(* CODESYS project plc_chalet_xts.library
   Title: CHALET_Xts
   Version: 4.0.4
   Placeholder: CHALET_Xts
   Company: Beckhoff CH

Project tree, tasks and I/O mapping:
  libraries: CHALET_BaseComponents, * (Beckhoff CH); CHALET_Nc, * (Beckhoff CH); Tc2_EtherCAT, * (Beckhoff Automation GmbH); Tc2_Math, * (Beckhoff Automation GmbH); Tc2_MC2, * (Beckhoff Automation GmbH); Tc2_Standard, * (Beckhoff Automation GmbH); Tc2_System, * (Beckhoff Automation GmbH); Tc3_EventLogger, * (Beckhoff Automation GmbH); Tc3_Mc3Definitions, * (Beckhoff Automation GmbH); Tc3_McCollisionAvoidance, * (Beckhoff Automation GmbH); Tc3_McCoordinatedMotion, * (Beckhoff Automation GmbH); Tc3_Module, * (Beckhoff Automation GmbH); Tc3_XTS_Utility, * (Beckhoff Automation GmbH)
  COMPENENTs/
    Casting/
      function ToEnvironment [ST]
      function ToGroup [ST]
      function ToMover [ST]
      function ToMover_PLC [ST]
      function ToStation [ST]
      function ToStation_PLC [ST]
      function ToTrigger [ST]
    Environment/
      function block FB_XTS_Environment [ST]: FB_init, HR, Initialize, TrackIsRing, TrackLength, Update, UtilityEnvirement
      interface I_XTS_Environment: HR, Initialize, TrackIsRing, TrackLength, Update, UtilityEnvirement
    Group/
      data type E_NcGroupCommands
      function block FB_XTS_Group [ST]: AddAxisListToGroup, AddingAxisToGroup, AllAxesStanding, ChangeGapMode, Disable, Enable, FB_init, GroupEnabled, HR, Initialize, Mapped, OID, RemoveAxisFromGroup, Reset, UngroupAllAxes, Update, UtilityCAGroup
      interface I_XTS_Group: AddAxisListToGroup, AddingAxisToGroup, AllAxesStanding, ChangeGapMode, Disable, Enable, GroupEnabled, HR, Initialize, RemoveAxisFromGroup, Reset, UngroupAllAxes, Update, UtilityCAGroup
    Mover/
      ProductData/
        function block FB_XTS_ProductData [ST]: LinkedMover, LinkToMover
        interface I_XTS_ProductData: LinkedMover, LinkToMover
      function block FB_XTS_Axis [ST]: HaltCA, MoveAbsoluteCA, Update
      function block FB_XTS_Mover [ST]: Disable, Enable, HaltCA, MoveAbsCA, Reset, DefaultAcceleration, DefaultDeceleration, DefaultJerk, SetAcceleration, SetVelocity, Coupled, DrivenDistance, Feedback, getAxisRef, IdentInGroup, LagDistance, LastCmdTargedGap, LastCmdTargedPosition, LastCmdTargedVelocity, MoverInGroup, Moving, NextMover, OID, ParentStation, PositionOnTrack, TargedStation, FB_init, FullAccess, Initialize, ProductData, Update, UtilityMover
      interface I_XTS_Mover: Coupled, Disable, DrivenDistance, Enable, Feedback, getAxisRef, HaltCA, IdentInGroup, LagDistance, LastCmdTargedGap, LastCmdTargedPosition, LastCmdTargedVelocity, MoveAbsCA, MoverInGroup, Moving, NextMover, OID, ParentStation, PositionOnTrack, Reset, SetAcceleration, SetVelocity, TargedStation, UtilityMover
      interface I_XTS_Mover_PLC: DefaultAcceleration, DefaultDeceleration, DefaultJerk, DrivenDistance, FullAccess, LagDistance, LastCmdTargedGap, LUID, PositionOnTrack, ProductData, SetVelocity, TargedStation, UtilityMover
    Station/
      function block FB_XTS_Station [ST]: ChangePos, CtsEmptySpaceInQueue, CtsMoversInQueue, FullAccess, MoverGapAtExit, MoverQueueSize, MoversInPlace, MoversInQueue, MoverVelocityAtExit, PositionOnTrack, SuppressDynamicsChange, TargetPosMonitoringTime, TargetPosWindow, ProcessSimulationActive, Simulation, SimulationMode, MoverPerMin, UpdateStatistic, UpdateUtilityStation, UtilityStationInfo, AddMoverToQueue, DeleteMoversQueue, FB_init, HR, Initialize, OID, Prepare, ReadyToRecvMovers, SendMoversToStation, StationBehinde, StationsAhead, TrySendMoverToNextStation, Update
      interface I_XTS_Station: AddMoverToQueue, CtsEmptySpaceInQueue, CtsMoversInQueue, DeleteMoversQueue, HR, LUID, MoverGapAtExit, MoverQueueSize, MoversInPlace, MoversInQueue, MoverVelocityAtExit, PositionOnTrack, ReadyToRecvMovers, SendMoversToStation, StationsAhead
      interface I_XTS_Station_PLC: ProcessSimulationActive, SimulationMode, ChangePos, FullAccess, LUID, MoverQueueSize, MoversInPlace, MoversInQueue, MoverVelocityAtExit, PositionOnTrack, ReadyToRecvMovers, SendMoversToStation, SuppressDynamicsChange, TargetPosMonitoringTime, TargetPosWindow
    System/
      function block FB_XTS_System [ST]: Disable, Disabled, Disabling, Enable, Enabled, Enabling, Initialize, Initialized, LinkEnvironment, LinkGroup, RegisterMover, RegisterStation, RegisterTrigger, RegisterZone, Environment, Feedback, getMoverInFront, getStationInFront, Movers, Reset, Station, Stations, SuppressAllDynamicsChanges, TrackLength, Triggers, Update, Zones
      interface I_XTS_System_PLC: Disable, Disabled, Enable, Enabled, Feedback, Initialize, Initialized, Reset, Station, SuppressAllDynamicsChanges, TrackLength, Update
      interface I_XTS_System_Registration: Disabled, Enabled, Environment, getMoverInFront, getStationInFront, Initialized, LinkEnvironment, LinkGroup, Movers, RegisterMover, RegisterStation, RegisterTrigger, RegisterZone, Stations, TrackLength
    Trigger/
      function block FB_XTS_Trigger [ST]: FB_init, HR, Initialize, ListOfMoversToCheck, MoverAtTrigger, MoverDetected, PositionOnTrack, Prepare, TimeStamp, TriggerDirection, Update
      interface I_XTS_Trigger: HR, ListOfMoversToCheck, MoverAtTrigger, MoverDetected, PositionOnTrack, TimeStamp, TriggerDirection
    Zone/
      function block FB_XTS_Zone [ST]: CtsMoversInZone, EndPositionOnTrack, FB_init, HR, Initialize, ListOfMoversToCheck, MoversInZone, Prepare, StartPositionOnTrack, Update
      interface I_XTS_Zone: CtsMoversInZone, EndPositionOnTrack, HR, ListOfMoversToCheck, MoversInZone, StartPositionOnTrack
    Class Diagram
  Diag/
    function block FB_XtsEtherCatDiag [ST]: FB_init, Initialize, Initialized, Update
    data type ST_XtsMotorEtherCatDiag
  FUNCTIONs/
    function F_BuildLogString [ST]
    function F_GetDistToPosModulo [ST]
    function F_InLimitTest [ST]
  00000000-0000-0000-0000-000000000000|LICENSE.md
  LICENSE.md
  global variables XtsParameterlist
*)

// COMPENENTs/Group/E_NcGroupCommands
{attribute 'qualified_only'}
{attribute 'strict'}
{attribute 'to_string'}
TYPE E_NcGroupCommands :
(
	None:=0,
	GroupDisable:=150,
	GroupEnable,
	GroupReset,
	AddAxisListToGroup,
	RemoveAxisFromGroup,
	UngroupAllAxes
);
END_TYPE

// Diag/ST_XtsMotorEtherCatDiag
TYPE ST_XtsMotorEtherCatDiag :
STRUCT
	fbSource : FB_TcSourceInfo;
	fbAlarmNotInOpMode : FB_TcAlarm;
	fbAlarmNoCommunication : FB_TcAlarm;
	
	fbGetSlaveState : FB_EcGetSlaveState;
	nLastState : BYTE;
END_STRUCT
END_TYPE

// XtsParameterlist
{attribute 'qualified_only'}
VAR_GLOBAL CONSTANT
	
	(*Checks whether the TC3 event logger is set as standard in the XTS prosessing unit.*)
	B_MSG_IF_TC3EVENTLOGGER_IS_NOT_DEFAULT: BOOL := TRUE;	

	MAX_MOVER_PER_SYSTEM : UINT := 50;
	MAX_MOTORS_PER_SYSTEM : UINT := 100;
	STATISTIC_AVG_PERIOD : TIME := T#10S;
END_VAR

// COMPENENTs/Casting/ToEnvironment
FUNCTION ToEnvironment : BOOL
VAR_INPUT
	ipChObject : I_CH_OBJECT;
	ipXtsEnvironment : REFERENCE TO I_XTS_Environment;
END_VAR

VAR
	ipTmp : I_XTS_Environment;
END_VAR

(* 
   1. Test if the interface exists
   2. Test if the object implements a "Object" interface 
   3. Write reference to interface in parameter
   4. Returne TRUE if succesfull
*)
IF ipChObject <> 0 AND_THEN __QUERYINTERFACE(ipChObject,ipTmp) THEN
	ipXtsEnvironment := ipTmp;
	ToEnvironment := TRUE;
END_IF

END_FUNCTION

// COMPENENTs/Environment/I_XTS_Environment
INTERFACE I_XTS_Environment  EXTENDS I_CH_Object

{attribute 'monitoring':='call'}
PROPERTY HR : HRESULT
GET
END_GET
END_PROPERTY

METHOD Initialize : HRESULT
END_METHOD

{attribute 'monitoring':='call'}
PROPERTY TrackIsRing : BOOL
GET
END_GET
END_PROPERTY

{attribute 'monitoring':='call'}
PROPERTY TrackLength : LREAL
GET
END_GET
END_PROPERTY

METHOD Update : HRESULT
VAR_INPUT
END_VAR
END_METHOD

PROPERTY UtilityEnvirement : Tc3_XTS_Utility.i_TcIoXtsEnvironment
GET
END_GET
END_PROPERTY

END_INTERFACE

// COMPENENTs/Casting/ToGroup
FUNCTION ToGroup : BOOL
VAR_INPUT
	ipChObject : I_CH_OBJECT;
	ipXtsGroup : REFERENCE TO I_XTS_Group;
END_VAR

VAR
	ipTmp : I_XTS_Group;
END_VAR

(* 
   1. Test if the interface exists
   2. Test if the object implements a "Object" interface 
   3. Write reference to interface in parameter
   4. Returne TRUE if succesfull
*)
IF ipChObject <> 0 AND_THEN __QUERYINTERFACE(ipChObject,ipTmp) THEN
	ipXtsGroup := ipTmp;
	ToGroup := TRUE;
END_IF

END_FUNCTION

// COMPENENTs/Group/I_XTS_Group
INTERFACE I_XTS_Group  EXTENDS I_CH_Object

METHOD AddAxisListToGroup : HRESULT
VAR_INPUT
	ipMovers : I_CH_List;
END_VAR
END_METHOD

METHOD AddingAxisToGroup : HRESULT
END_METHOD

PROPERTY AllAxesStanding : Bool
GET
END_GET
END_PROPERTY

METHOD ChangeGapMode : HRESULT
VAR_INPUT
	bFast : BOOL;
END_VAR
END_METHOD

METHOD Disable : HRESULT
VAR_INPUT
END_VAR
END_METHOD

METHOD Enable : HRESULT
VAR_INPUT
END_VAR
END_METHOD

{attribute 'monitoring':='call'}
PROPERTY GroupEnabled : BOOL
GET
END_GET
END_PROPERTY

{attribute 'monitoring':='call'}
PROPERTY HR : HRESULT
GET
END_GET
END_PROPERTY

METHOD Initialize : HRESULT
VAR_INPUT
END_VAR
END_METHOD

METHOD RemoveAxisFromGroup : HRESULT
VAR_INPUT
	ipMover : I_XTS_Mover;
END_VAR
END_METHOD

METHOD Reset : HRESULT
VAR_INPUT
END_VAR
END_METHOD

METHOD UngroupAllAxes : HRESULT
VAR_INPUT
END_VAR
END_METHOD

METHOD Update : HRESULT
VAR_INPUT
END_VAR
END_METHOD

{attribute 'monitoring':='call'}
PROPERTY UtilityCAGroup : I_Mc2CaGroup
GET
END_GET
END_PROPERTY

END_INTERFACE

// COMPENENTs/Mover/I_XTS_Mover
INTERFACE I_XTS_Mover EXTENDS I_CH_Object

{attribute 'OPC.UA.DA.Property' := '1'}
{attribute 'monitoring':='call'}
PROPERTY Coupled : BOOL
GET
END_GET
END_PROPERTY

METHOD Disable : HRESULT
VAR_INPUT
END_VAR
END_METHOD

{attribute 'monitoring':='call'}
PROPERTY DrivenDistance : LREAL
GET
END_GET
END_PROPERTY

METHOD Enable : HRESULT
VAR_INPUT
END_VAR
END_METHOD

{attribute 'OPC.UA.DA.Property' := '1'}
{attribute 'monitoring':='call'}
PROPERTY Feedback : I_CH_Feedback
GET
END_GET
END_PROPERTY

PROPERTY getAxisRef : REFERENCE TO Tc2_MC2.AXIS_REF
GET
END_GET
END_PROPERTY

METHOD HaltCA : HRESULT
VAR_INPUT
END_VAR
END_METHOD

{attribute 'monitoring':='call'}
PROPERTY IdentInGroup : IDENT_IN_GROUP_REF
GET
END_GET
END_PROPERTY

{attribute 'monitoring':='call'}
PROPERTY LagDistance : LREAL
GET
END_GET
END_PROPERTY

{attribute 'monitoring':='call'}
PROPERTY LastCmdTargedGap : LREAL
GET
END_GET
END_PROPERTY

{attribute 'monitoring':='call'}
PROPERTY LastCmdTargedPosition : LREAL
GET
END_GET
END_PROPERTY

{attribute 'monitoring':='call'}
PROPERTY LastCmdTargedVelocity : LREAL
GET
END_GET
END_PROPERTY

METHOD MoveAbsCA : HRESULT
VAR_INPUT
    fPosition              : LREAL;
    fVelocity              : LREAL;
    fGap                   : LREAL;
    eDirection             : Tc3_Mc3Definitions.MC_DIRECTION;
END_VAR
END_METHOD

{attribute 'monitoring':='call'}
PROPERTY MoverInGroup : BOOL
GET
END_GET
SET
END_SET
END_PROPERTY

{attribute 'OPC.UA.DA.Property' := '1'}
{attribute 'monitoring':='call'}
PROPERTY Moving : BOOL
GET
END_GET
END_PROPERTY

{attribute 'monitoring':='call'}
PROPERTY NextMover : I_XTS_Mover
GET
END_GET
END_PROPERTY

{attribute 'monitoring':='call'}
PROPERTY OID : OTCID
GET
END_GET
END_PROPERTY

{attribute 'monitoring':='call'}
PROPERTY ParentStation : I_XTS_Station
GET
END_GET
SET
END_SET
END_PROPERTY

{attribute 'monitoring':='call'}
PROPERTY PositionOnTrack : LREAL
GET
END_GET
END_PROPERTY

METHOD Reset : HRESULT
VAR_INPUT
END_VAR
END_METHOD

{attribute 'monitoring':='call'}
PROPERTY SetAcceleration : LREAL
GET
END_GET
END_PROPERTY

{attribute 'monitoring':='call'}
PROPERTY SetVelocity : LREAL
GET
END_GET
END_PROPERTY

{attribute 'monitoring':='call'}
PROPERTY TargedStation : STRING
GET
END_GET
SET
END_SET
END_PROPERTY

{attribute 'monitoring':='call'}
PROPERTY UtilityMover : I_TcIoXtsXpuMover
GET
END_GET
END_PROPERTY

END_INTERFACE

// COMPENENTs/Station/I_XTS_Station
INTERFACE I_XTS_Station EXTENDS I_CH_Object

METHOD AddMoverToQueue : HRESULT
VAR_INPUT
	ipMover : I_XTS_Mover;
END_VAR
END_METHOD

{attribute 'monitoring':='call'}
PROPERTY CtsEmptySpaceInQueue : UDINT
GET
END_GET
END_PROPERTY

{attribute 'monitoring':='call'}
PROPERTY CtsMoversInQueue : UDINT
GET
END_GET
END_PROPERTY

METHOD DeleteMoversQueue : HRESULT
VAR_INPUT
END_VAR
END_METHOD

{attribute 'monitoring':='call'}
PROPERTY HR : HRESULT
GET
END_GET
END_PROPERTY

{attribute 'monitoring':='call'}
PROPERTY LUID : STRING
GET
END_GET
END_PROPERTY

{attribute 'monitoring':='call'}
PROPERTY MoverGapAtExit : LREAL
GET
END_GET
END_PROPERTY

{attribute 'monitoring':='call'}
PROPERTY MoverQueueSize : UINT
GET
END_GET
SET
END_SET
END_PROPERTY

{attribute 'monitoring':='call'}
PROPERTY MoversInPlace : BOOL
GET
END_GET
END_PROPERTY

{attribute 'monitoring':='call'}
PROPERTY MoversInQueue : REFERENCE TO ARRAY [0..(XtsParameterlist.MAX_MOVER_PER_SYSTEM-1)] OF I_XTS_Mover_PLC // Return a sorted list of movers in this zone. Index 0 is the mover in Front.
GET
END_GET
END_PROPERTY

{attribute 'monitoring':='call'}
PROPERTY MoverVelocityAtExit : LREAL
GET
END_GET
SET
END_SET
END_PROPERTY

{attribute 'monitoring':='call'}
PROPERTY PositionOnTrack : LREAL
GET
END_GET
END_PROPERTY

{attribute 'monitoring':='call'}
PROPERTY ReadyToRecvMovers : BOOL
GET
END_GET
SET
END_SET
END_PROPERTY

METHOD SendMoversToStation : HRESULT
VAR_INPUT
	sTargedStation : STRING;
END_VAR
END_METHOD

{attribute 'monitoring':='call'}
PROPERTY StationsAhead : I_XTS_Station
GET
END_GET
END_PROPERTY

END_INTERFACE

// COMPENENTs/Mover/I_XTS_Mover_PLC
INTERFACE I_XTS_Mover_PLC EXTENDS I_CH_Object

{attribute 'OPC.UA.DA.Property' := '1'}
{attribute 'monitoring':='call'}
PROPERTY DefaultAcceleration : LREAL
GET
END_GET
SET
END_SET
END_PROPERTY

{attribute 'OPC.UA.DA.Property' := '1'}
{attribute 'monitoring':='call'}
PROPERTY DefaultDeceleration : LREAL
GET
END_GET
SET
END_SET
END_PROPERTY

{attribute 'OPC.UA.DA.Property' := '1'}
{attribute 'monitoring':='call'}
PROPERTY DefaultJerk : LREAL
GET
END_GET
SET
END_SET
END_PROPERTY

{attribute 'monitoring':='call'}
PROPERTY DrivenDistance : LREAL
GET
END_GET
END_PROPERTY

(*The _ PLC interface provides the user with a simplified interface for commanding between the stations. Sometimes, however, this is not enough. 
Either you get the corresponding interface with the __Queryinterface or you can get full access with this property.*)
PROPERTY FullAccess : I_XTS_Mover
GET
END_GET
END_PROPERTY

{attribute 'monitoring':='call'}
PROPERTY LagDistance : LREAL
GET
END_GET
END_PROPERTY

{attribute 'monitoring':='call'}
PROPERTY LastCmdTargedGap : LREAL
GET
END_GET
END_PROPERTY

{attribute 'monitoring':='call'}
PROPERTY LUID : STRING
GET
END_GET
END_PROPERTY

{attribute 'monitoring':='call'}
PROPERTY PositionOnTrack : LREAL
GET
END_GET
END_PROPERTY

{attribute 'monitoring':='call'}
PROPERTY PUBLIC ProductData : I_XTS_ProductData
GET
END_GET
SET
END_SET
END_PROPERTY

{attribute 'monitoring':='call'}
PROPERTY SetVelocity : LREAL
GET
END_GET
END_PROPERTY

{attribute 'monitoring':='call'}
PROPERTY TargedStation : STRING
GET
END_GET
END_PROPERTY

{attribute 'monitoring':='call'}
PROPERTY UtilityMover : I_TcIoXtsXpuMover
GET
END_GET
END_PROPERTY

END_INTERFACE

// COMPENENTs/Mover/ProductData/I_XTS_ProductData
INTERFACE I_XTS_ProductData EXTENDS __SYSTEM.IQueryInterface

{attribute 'monitoring':='call'}
PROPERTY LinkedMover : I_XTS_Mover_PLC
GET
END_GET
END_PROPERTY

METHOD LinkToMover : BOOL //it is not necessary to call this method. This is already done internally
VAR_INPUT
	ipMoverPlc : I_XTS_Mover_PLC;
END_VAR
END_METHOD

END_INTERFACE

// COMPENENTs/Casting/ToMover
FUNCTION ToMover : BOOL
VAR_INPUT
	ipChObject : I_CH_OBJECT;
	ipXtsMover : REFERENCE TO I_XTS_Mover;
END_VAR

VAR
	ipTmp : I_XTS_Mover;
END_VAR

(* 
   1. Test if the interface exists
   2. Test if the object implements a "Object" interface 
   3. Write reference to interface in parameter
   4. Returne TRUE if succesfull
*)
IF ipChObject <> 0 AND_THEN __QUERYINTERFACE(ipChObject,ipTmp) THEN
	ipXtsMover := ipTmp;
	ToMover := TRUE;
END_IF

END_FUNCTION

// COMPENENTs/Casting/ToMover_PLC
FUNCTION ToMover_PLC : BOOL
VAR_INPUT
	ipChObject : I_CH_OBJECT;
	ipXtsMover : REFERENCE TO I_XTS_Mover_PLC;
END_VAR

VAR
	ipTmp : I_XTS_Mover_PLC;
END_VAR

(* 
   1. Test if the interface exists
   2. Test if the object implements a "Object" interface 
   3. Write reference to interface in parameter
   4. Returne TRUE if succesfull
*)
IF ipChObject <> 0 AND_THEN __QUERYINTERFACE(ipChObject,ipTmp) THEN
	ipXtsMover := ipTmp;
	ToMover_PLC := TRUE;
END_IF

END_FUNCTION

// COMPENENTs/Casting/ToStation
FUNCTION ToStation : BOOL
VAR_INPUT
	ipChObject : I_CH_OBJECT;
	ipXtsStation : REFERENCE TO I_XTS_Station;
END_VAR

VAR
	ipTmp : I_XTS_Station;
END_VAR

(* Register the Station
   1. Test if the interface exists
   2. Test if the object implements a "Object" interface 
*)
IF ipChObject <> 0 AND_THEN __QUERYINTERFACE(ipChObject,ipTmp) THEN
	ipXtsStation := ipTmp;
	ToStation := TRUE;
END_IF

END_FUNCTION

// COMPENENTs/Casting/ToStation_PLC
FUNCTION ToStation_PLC : BOOL
VAR_INPUT
	ipChObject : I_CH_OBJECT;
	ipXtsStationPLC : REFERENCE TO I_XTS_Station_PLC;
END_VAR

VAR
	ipTmp : I_XTS_Station_PLC;
END_VAR

(* Register the Station
   1. Test if the interface exists
   2. Test if the object implements a "Object" interface 
*)
IF ipChObject <> 0 AND_THEN __QUERYINTERFACE(ipChObject,ipTmp) THEN
	ipXtsStationPLC := ipTmp;
	ToStation_PLC := TRUE;
END_IF

END_FUNCTION

// COMPENENTs/Station/I_XTS_Station_PLC
INTERFACE I_XTS_Station_PLC EXTENDS I_CH_Object

{attribute 'monitoring':='call'}
PROPERTY ProcessSimulationActive : BOOL
GET
END_GET
END_PROPERTY

//If a valid time (>0seconds) is set and the configured destination station exists, then the movers will be sent away automatically after this time from now on.
METHOD SimulationMode : HRESULT
VAR_INPUT
	fProcessDuration 	: LREAL; //[s]
	sTargedStation		: STRING; //LUID of the targed station to automatic send after the duration
END_VAR
END_METHOD

METHOD ChangePos : HRESULT
VAR_INPUT
	fNewPosOnTrack : LREAL;
END_VAR
END_METHOD

(*The _ PLC interface provides the user with a simplified interface for commanding between the stations. Sometimes, however, this is not enough. 
Either you get the corresponding interface with the __Queryinterface or you can get full access with this property.*)
PROPERTY FullAccess : I_XTS_Station
GET
END_GET
END_PROPERTY

{attribute 'monitoring':='call'}
PROPERTY LUID : STRING
GET
END_GET
END_PROPERTY

{attribute 'monitoring':='call'}
PROPERTY MoverQueueSize : UINT
GET
END_GET
SET
END_SET
END_PROPERTY

{attribute 'monitoring':='call'}
PROPERTY MoversInPlace : BOOL
GET
END_GET
END_PROPERTY

{attribute 'monitoring':='call'}
PROPERTY MoversInQueue : REFERENCE TO ARRAY [0..(XtsParameterlist.MAX_MOVER_PER_SYSTEM-1)] OF I_XTS_Mover_PLC // Return a sorted list of movers in this zone. Index 0 is the mover in Front.
GET
END_GET
END_PROPERTY

{attribute 'monitoring':='call'}
PROPERTY MoverVelocityAtExit : LREAL //[mm/s] Every mover that leaves or passes the station gets this new velocity as a target.
GET
END_GET
SET
END_SET
END_PROPERTY

{attribute 'monitoring':='call'}
PROPERTY PositionOnTrack : LREAL
GET
END_GET
END_PROPERTY

{attribute 'monitoring':='call'}
//prevent further movers from entering the station, 
//e.g. to prevent a collision. All movers that are already moving to reach this station will be stopped with a stop 
//and restarted with Ready True.
PROPERTY ReadyToRecvMovers : BOOL
GET
END_GET
SET
END_SET
END_PROPERTY

METHOD SendMoversToStation : HRESULT
VAR_INPUT
	sTargedStation : STRING;
END_VAR
END_METHOD

{attribute 'monitoring':='call'}
PROPERTY SuppressDynamicsChange : BOOL
GET
END_GET
SET
END_SET
END_PROPERTY

{attribute 'monitoring':='call'}
//A time that is waited as soon as the mover is in the station (including the monitoring window) before “MoversInPlace” is set. e.g. used to stabilize the workpiece
PROPERTY TargetPosMonitoringTime : TIME
GET
END_GET
SET
END_SET
END_PROPERTY

{attribute 'monitoring':='call'}
//How many mm before the mover reaches the position is “MoversInPlace” set for the process. 
//This distance can also be set very large (e.g. 100mm) for moving past without stopping.
PROPERTY TargetPosWindow : LREAL
GET
END_GET
SET
END_SET
END_PROPERTY

END_INTERFACE

// COMPENENTs/Casting/ToTrigger
FUNCTION ToTrigger : BOOL
VAR_INPUT
	ipChObject : I_CH_OBJECT;
	ipXtsTrigger : REFERENCE TO I_XTS_Trigger;
END_VAR

VAR
	ipTmp : I_XTS_Trigger;
END_VAR

(* 
   1. Test if the interface exists
   2. Test if the object implements a "Object" interface 
   3. Write reference to interface in parameter
   4. Returne TRUE if succesfull
*)
IF ipChObject <> 0 AND_THEN __QUERYINTERFACE(ipChObject,ipTmp) THEN
	ipXtsTrigger := ipTmp;
	ToTrigger := TRUE;
END_IF

END_FUNCTION

// COMPENENTs/Trigger/I_XTS_Trigger
INTERFACE I_XTS_Trigger  EXTENDS I_CH_Object

{attribute 'monitoring':='call'}
PROPERTY HR : HRESULT
GET
END_GET
END_PROPERTY

PROPERTY ListOfMoversToCheck : I_CH_List
SET
END_SET
END_PROPERTY

{attribute 'monitoring':='call'}
PROPERTY MoverAtTrigger : I_XTS_Mover
GET
END_GET
END_PROPERTY

{attribute 'monitoring':='call'}
PROPERTY MoverDetected : BOOL
GET
END_GET
END_PROPERTY

{attribute 'monitoring':='call'}
PROPERTY PositionOnTrack : LREAL
GET
END_GET
SET
END_SET
END_PROPERTY

{attribute 'monitoring':='call'}
PROPERTY TimeStamp : T_DCTIME64;
GET
END_GET
END_PROPERTY

{attribute 'monitoring':='call'}
PROPERTY TriggerDirection : Tc2_MC2.MC_Direction
GET
END_GET
SET
END_SET
END_PROPERTY

END_INTERFACE

// COMPENENTs/Environment/FB_XTS_Environment
{attribute 'no_explicit_call' := 'Do not call the body - Stick to OOP'}
FUNCTION_BLOCK FB_XTS_Environment EXTENDS FB_CH_Object IMPLEMENTS I_XTS_Environment
VAR
	{attribute 'hide'}
	bInitDone : BOOL ;
	{attribute 'hide'}
	ipXtsSystem : I_XTS_System_Registration;

	fbUtilityEnvironment : Tc3_XTS_Utility.FB_TcIoXtsEnvironment;
	
	//Ethercat Diagnostic of all XTS Motors
	fbXtsEtherCatDiag		: FB_XtsEtherCatDiag(	ipUtilityEnvironmentv 				:=  fbUtilityEnvironment,
													bCheckIfTc3EventloggerIsSelected 	:= XtsParameterlist.B_MSG_IF_TC3EVENTLOGGER_IS_NOT_DEFAULT);
	
	{attribute 'hide'}
	fbXtsEnvironmentVisu : Tc3_XTS_Utility.FB_XtsEnvironmentVisu;
		
END_VAR

METHOD FB_init : BOOL
VAR_INPUT
	bInitRetains : BOOL; // if TRUE, the retain variables are initialized (warm start / cold start)
	bInCopyCode : BOOL;  // if TRUE, the instance afterwards gets moved into the copy code (online change)

	ipXtsSystem : I_XTS_System_Registration; //Interface to XTS system object	
END_VAR
VAR_INST
	{attribute 'hide'}
	bFBInitCalledOnce : BOOL; //Do the following code once during start up and not during onlinechange
END_VAR
//Do the following code once during start up and not during onlinechange
IF NOT bFBInitCalledOnce THEN 
	
	//Regristrate object in System
	IF ipXtsSystem <> 0 THEN
		ipXtsSystem.LinkEnvironment(THIS^);
		THIS^.ipXtsSystem := ipXtsSystem;
	END_IF



END_IF

bFBInitCalledOnce := TRUE;
END_METHOD

{warning 'add property implementation'}
{attribute 'monitoring':='call'}
PROPERTY HR : HRESULT
GET
HR := S_OK;
END_GET
END_PROPERTY

METHOD Initialize : HRESULT
VAR 
	hr : HRESULT;
END_VAR
IF NOT THIS^.bInitDone THEN
	Initialize := S_PENDING;	

	//Enable init Info Server if needed
	fbUtilityEnvironment.P_XtsEnvironmentConfiguration.bEnableInitInfoServer := TRUE;

	//Enable init CA Group if needed
	fbUtilityEnvironment.P_XtsEnvironmentConfiguration.bEnableInitCaGroup := TRUE;

	IF NOT fbUtilityEnvironment.P_IsInitialized THEN	
		//Start init
		fbUtilityEnvironment.Init(bExecute := TRUE); 
		hr := GetMostSignificant(hr, S_PENDING);	
 	ELSE
		//Stop init
		fbUtilityEnvironment.Init(bExecute := FALSE);
	END_IF
	
	// Link data Pointer 
	fbXtsEnvironmentVisu(ipTcIoXtsEnvironment:=UtilityEnvirement);

	// Ethercat Diagnostic of all XTS Motors
	hr := GetMostSignificant(hr, fbXtsEtherCatDiag.Initialize());
	

	THIS^.bInitDone  :=  hr = S_OK;
END_IF

Initialize := hr;
END_METHOD

{attribute 'monitoring':='call'}
PROPERTY TrackIsRing : BOOL
GET
IF fbUtilityEnvironment.P_IsInitialized THEN
	TrackIsRing := fbUtilityEnvironment.Mc2CaGroup(1).GetRailIsRing();
END_IF
END_GET
END_PROPERTY

{attribute 'monitoring':='call'}
PROPERTY TrackLength : LREAL
GET
IF fbUtilityEnvironment.P_IsInitialized THEN
	TrackLength := fbUtilityEnvironment.Mc2CaGroup(1).GetRailLength();
END_IF
END_GET
END_PROPERTY

METHOD Update : HRESULT
VAR
	hr : HRESULT;
END_VAR

fbXtsEtherCatDiag.Update();

fbXtsEnvironmentVisu.Cycle();

Update:= hr;
END_METHOD

PROPERTY UtilityEnvirement : Tc3_XTS_Utility.I_TcIoXtsEnvironment
GET
//Interface to envirement
UtilityEnvirement := fbUtilityEnvironment;
END_GET
END_PROPERTY

END_FUNCTION_BLOCK

// COMPENENTs/System/I_XTS_System_Registration
INTERFACE I_XTS_System_Registration

{attribute 'monitoring':='call'}
PROPERTY Disabled : Bool
GET
END_GET
END_PROPERTY

{attribute 'monitoring':='call'}
PROPERTY Enabled : Bool
GET
END_GET
END_PROPERTY

{attribute 'monitoring':='call'}
PROPERTY Environment : I_XTS_Environment
GET
END_GET
END_PROPERTY

METHOD getMoverInFront : I_Xts_Mover
VAR_INPUT
	ipMover : I_Xts_Mover;
END_VAR
END_METHOD

METHOD getStationInFront : I_XTS_Station
VAR_INPUT
	ipStation : I_XTS_Station;
END_VAR
END_METHOD

{attribute 'monitoring':='call'}
PROPERTY Initialized : BOOL
GET
END_GET
END_PROPERTY

METHOD LinkEnvironment : HRESULT
VAR_INPUT
	ipEnvironment : CHALET_BaseComponents.I_CH_Object;
END_VAR
END_METHOD

METHOD LinkGroup : HRESULT
VAR_INPUT
	ipGroup : CHALET_BaseComponents.I_CH_Object;
END_VAR
END_METHOD

{attribute 'monitoring':='call'}
PROPERTY Movers : CHALET_BaseComponents.I_CH_LIST
GET
END_GET
END_PROPERTY

METHOD RegisterMover : HRESULT
VAR_INPUT
	ipMover : CHALET_BaseComponents.I_CH_Object;
END_VAR
END_METHOD

METHOD RegisterStation : HRESULT
VAR_INPUT
	ipStation : CHALET_BaseComponents.I_CH_Object;
END_VAR
END_METHOD

METHOD RegisterTrigger : HRESULT
VAR_INPUT
	ipTrigger	: CHALET_BaseComponents.I_CH_Object;
END_VAR
END_METHOD

METHOD RegisterZone : HRESULT
VAR_INPUT
	ipZone	: CHALET_BaseComponents.I_CH_Object;
END_VAR
END_METHOD

PROPERTY Stations : I_CH_LIST
GET
END_GET
END_PROPERTY

{attribute 'monitoring':='call'}
PROPERTY TrackLength : LREAL
GET
END_GET
END_PROPERTY

END_INTERFACE

// Diag/FB_XtsEtherCatDiag
{attribute 'no_explicit_call' := 'Do not call the body - Stick to OOP'}
(* This FB generates an array with all XTS motor modules. These are now checked cyclically one after the other to see whether the EtherCAT slave controller is in OP mode *)
FUNCTION_BLOCK FB_XtsEtherCatDiag EXTENDS CHALET_BaseComponents.FB_CH_Object
VAR
	ipUtilityEnvironmentv : Tc3_XTS_Utility.I_TcIoXtsEnvironment;
	bCheckIfTc3EventloggerIsSelected : BOOL;
	stMotorDiag : ARRAY[0..N_MAX_CTS_MOTORMODULES-1] OF ST_XtsMotorEtherCatDiag;
	bInitDone : BOOL;
	nIdxTrigger : UINT;
	nCtnMotorModules : UINT;
	fbMsgWrongEventlogger : FB_TcMessage;
	bEventLoggerChecked : BOOL;
END_VAR

VAR CONSTANT
	N_MAX_CTS_MOTORMODULES : UINT := XtsParameterlist.MAX_MOTORS_PER_SYSTEM;
END_VAR

METHOD FB_init : BOOL
VAR_INPUT
	bInitRetains : BOOL; // if TRUE, the retain variables are initialized (warm start / cold start)
	bInCopyCode : BOOL;  // if TRUE, the instance afterwards gets moved into the copy code (online change)
	
	ipUtilityEnvironmentv : Tc3_XTS_Utility.I_TcIoXtsEnvironment;
	
	//Message if TC3_Eventlogger is not set as Eventlogger. Not possible to change online.
	//Must be adjusted in the following object: XtsProcessingUnit/Parameter(Init)/Diagnostic/UsedEventLogger 
	bCheckIfTc3EventloggerIsSelected : BOOL;
END_VAR

VAR
	fbGetCurTaskIdx  : GETCURTASKINDEX;
END_VAR

THIS^.ipUtilityEnvironmentv := ipUtilityEnvironmentv;
THIS^.bCheckIfTc3EventloggerIsSelected := bCheckIfTc3EventloggerIsSelected;
END_METHOD

METHOD Initialize : HRESULT
VAR
	ipObject : ITComObject;
	sObjectName : STRING;
	nIdx, nIdxXpu, nIdxPart, nIdxModule : UINT;
END_VAR
VAR_INST

END_VAR
//Validate interface
IF ipUtilityEnvironmentv = 0 THEN
	Initialize := E_FAIL;
	RETURN;
END_IF

//Wait for an valide XpuCount. At beginn, count is 0
IF ipUtilityEnvironmentv.P_XpuCount = 0 THEN
	Initialize := S_PENDING;;
	RETURN;
END_IF

//Wait for init done
FOR nIdxXpu := 1 TO TO_UINT(ipUtilityEnvironmentv.P_XpuCount)  DO
	IF NOT ipUtilityEnvironmentv.XpuTcIo(nIdxXpu).P_IsInitialized THEN
		Initialize := S_PENDING;;
		RETURN;
	END_IF
END_FOR

//Message if TC3_Eventlogger is not set as Eventlogger. Not possible to change online.
//Must be adjusted in the following object: XtsProcessingUnit/Parameter(Init)/Diagnostic/UsedEventLogger 
IF NOT bEventLoggerChecked  AND THIS^.bCheckIfTc3EventloggerIsSelected THEN
	FOR nIdxXpu := 1 TO TO_UINT(ipUtilityEnvironmentv.P_XpuCount) DO
		IF ipUtilityEnvironmentv.XpuTcIo(nIdxXpu).GetUsedEventLogger() <> EventMessenger.TC3EventLogger THEN
			fbMsgWrongEventlogger.CreateEx(stEventEntry:=TC_EVENTS.CHALET_XTS_Events.TC3EventloggerCheck, ipSourceInfo := THIS^.fbSourceInfo);
			fbMsgWrongEventlogger.Send(0);
			EXIT;
		END_IF
	END_FOR
END_IF
bEventLoggerChecked := TRUE;



//For all Modul in all Parts in all Processing-Units
nIdx := 0;
FOR nIdxXpu := 1 TO TO_UINT(ipUtilityEnvironmentv.P_XpuCount) DO
	FOR nIdxPart := 1 TO ipUtilityEnvironmentv.XpuTcIo(nIdxXpu).P_PartCount DO
		FOR nIdxModule := 1 TO ipUtilityEnvironmentv.XpuTcIo(nIdxXpu).PartTcIo(nIdxPart).P_ModuleCount DO
			//Error, array is to small
			IF (nIdx > (N_MAX_CTS_MOTORMODULES-1)) THEN
				Initialize := E_FAIL;
				RETURN;
			END_IF
			
			//Read object name of motor module
			FW_ObjMgr_GetObjectInstance(oid:= ipUtilityEnvironmentv.XpuTcIo(nIdxXpu).PartTcIo(nIdxPart).ModuleTcIo(nIdxModule).GetMotorTerminalOid() , iid:= TC_GLOBAL_IID_LIST.IID_ITComObject, pipUnk:= ADR(ipObject));
			//Read Name of object if interafce is valid
			IF ipObject <> 0 AND_THEN (ipObject.TcGetObjectName(ADR(sObjectName), SIZEOF(sObjectName)) = S_OK) THEN
				//Set source name + Modulename
				stMotorDiag[nIdx].fbSource.sName := '';
				stMotorDiag[nIdx].fbSource.ExtendName(sObjectName);
				stMotorDiag[nIdx].fbSource.ExtendName(' Part:');
				stMotorDiag[nIdx].fbSource.ExtendName(TO_STRING(nIdxPart));
				stMotorDiag[nIdx].fbSource.ExtendName(' Module:');
				stMotorDiag[nIdx].fbSource.ExtendName(TO_STRING(nIdxModule));	
				ipObject.TcRelease();
			ELSE
				//Set source name
				stMotorDiag[nIdx].fbSource.sName := '';
				stMotorDiag[nIdx].fbSource.ExtendName('Part:');
				stMotorDiag[nIdx].fbSource.ExtendName(TO_STRING(nIdxPart));
				stMotorDiag[nIdx].fbSource.ExtendName(' Module:');
				stMotorDiag[nIdx].fbSource.ExtendName(TO_STRING(nIdxModule));	
			END_IF
			

		
			//Create alarm
			stMotorDiag[nIdx].fbAlarmNotInOpMode.CreateEx(
					stEventEntry := TC_EVENTS.CHALET_XTS_Events.EtherCatSlaveNotInOpMode, 
					ipSourceInfo := stMotorDiag[nIdx].fbSource, 
					bWithConfirmation := FALSE);
					
			stMotorDiag[nIdx].fbAlarmNoCommunication.CreateEx(	
					stEventEntry:= TC_EVENTS.CHALET_XTS_Events.NoCommunication,
					ipSourceInfo 	:= stMotorDiag[nIdx].fbSource, 
					bWithConfirmation := FALSE);
					
			//store ADS conncetion info
			stMotorDiag[nIdx].fbGetSlaveState.sNetId := ipUtilityEnvironmentv.XpuTcIo(nIdxXpu).PartTcIo(nIdxPart).ModuleTcIo(nIdxModule).CoE.AmsNetId;
			stMotorDiag[nIdx].fbGetSlaveState.nSlaveAddr := ipUtilityEnvironmentv.XpuTcIo(nIdxXpu).PartTcIo(nIdxPart).ModuleTcIo(nIdxModule).GetDriveAddress();		

			nIdx := nIdx +1;	
			THIS^.nCtnMotorModules := nIdx;
		END_FOR
	END_FOR
END_FOR
bInitDone := TRUE;
Initialize := S_OK;;
END_METHOD

{attribute 'monitoring':='call'}
PROPERTY Initialized : BOOL
GET
Initialized := bInitDone;
END_GET
END_PROPERTY

METHOD Update : HRESULT
VAR
	nIdx : UINT;
	bErrorNoCom : BOOL;
	bInOpMode : BOOL;
	bReadOfStateFailed : BOOL;
END_VAR
// Force to do init
IF NOT THIS^.bInitDone THEN
	Initialize();
	RETURN;
END_IF


//Trigger each plc cycle 1 read of the motor ethercat slave state - if not allready busy
IF NOT stMotorDiag[nIdxTrigger].fbGetSlaveState.bBusy THEN
	stMotorDiag[nIdxTrigger].fbGetSlaveState(bExecute := TRUE);
	stMotorDiag[nIdxTrigger].fbGetSlaveState(bExecute := FALSE);
	nIdxTrigger := (nIdxTrigger + 1)MOD THIS^.nCtnMotorModules;
END_IF



//For all FBs
FOR nIdx := 0 TO (THIS^.nCtnMotorModules-1) DO
	(*	0x___1 = Slave in 'INIT' state
		0x___2 = Slave in 'PREOP' state
		0x___3 = Slave in 'BOOT' state
		0x___4 = Slave in 'SAFEOP' state
		0x___8 = Slave in 'OP' state		*)
		
		
	//Write Ethercat linkState in TC3 Eventlogger
	bErrorNoCom := (stMotorDiag[nIdx].fbGetSlaveState.state.linkState = 16#01(*NotPresent*));
	IF (NOT bErrorNoCom AND stMotorDiag[nIdx].fbAlarmNoCommunication.bRaised) THEN
		//No error - Reset	
		stMotorDiag[nIdx].fbAlarmNoCommunication.Clear(0,0);
	ELSIF (bErrorNoCom AND NOT stMotorDiag[nIdx].fbAlarmNoCommunication.bRaised) THEN
		//New Error - Raise
		stMotorDiag[nIdx].fbAlarmNoCommunication.ipArguments.Clear();
		stMotorDiag[nIdx].fbAlarmNoCommunication.Raise(0);
	ELSE
		//Alarm is already active
		;
	END_IF	

		
	//Re-Raise alarm on change of state if ethercatslave is not in OP-Mode - Clear if NoCommunication is raised
	bInOpMode := (stMotorDiag[nIdx].fbGetSlaveState.state.deviceState = 16#08(*OP*));
	bReadOfStateFailed := ((stMotorDiag[nIdx].fbGetSlaveState.state.deviceState AND 16#0F(*Mask values 0-15*)) = 16#00);
	IF ((bInOpMode OR bErrorNoCom OR bReadOfStateFailed) AND stMotorDiag[nIdx].fbAlarmNotInOpMode.bRaised) THEN
		//No error - Reset	
		stMotorDiag[nIdx].fbAlarmNotInOpMode.Clear(0,0);
		
	ELSIF (bInOpMode OR bErrorNoCom OR bReadOfStateFailed) THEN
		; //Do nothing
		
	ELSIF (stMotorDiag[nIdx].fbGetSlaveState.state.deviceState <> stMotorDiag[nIdx].nLastState) THEN
		//New Error - Reset, Create and Raise
		stMotorDiag[nIdx].fbAlarmNotInOpMode.Clear(0,0);
		CASE (stMotorDiag[nIdx].fbGetSlaveState.state.deviceState AND 16#0F(*Mask values 0-15*)) OF
			1:  stMotorDiag[nIdx].fbAlarmNotInOpMode.ipArguments.Clear().AddString('INIT'); 	
			2:  stMotorDiag[nIdx].fbAlarmNotInOpMode.ipArguments.Clear().AddString('PREOP');	
			3:  stMotorDiag[nIdx].fbAlarmNotInOpMode.ipArguments.Clear().AddString('BOOT');		
			4:  stMotorDiag[nIdx].fbAlarmNotInOpMode.ipArguments.Clear().AddString('SAFEOP');	
		END_CASE
		stMotorDiag[nIdx].fbAlarmNotInOpMode.Raise(0);
		
	ELSE
		//Alarm is already active
		;
	END_IF
	stMotorDiag[nIdx].nLastState := stMotorDiag[nIdx].fbGetSlaveState.state.deviceState;

	
	//Call cyclic fb
	stMotorDiag[nIdx].fbGetSlaveState();
END_FOR
END_METHOD

END_FUNCTION_BLOCK

// COMPENENTs/Group/FB_XTS_Group
{attribute 'no_explicit_call' := 'Do not call the body - Stick to OOP'}
FUNCTION_BLOCK FB_XTS_Group EXTENDS FB_CH_Object IMPLEMENTS I_XTS_Group
VAR
	{attribute 'hide'}	
	bInitDone : BOOL;
	{attribute 'hide'}
	ipXtsSystem 		: I_XTS_System_Registration;
	{attribute 'hide'}
	ipUtilityCAGroup 	: I_Mc2CaGroup;
	{attribute 'hide'}
	fbAddAxisToGroup 	: Tc3_McCoordinatedMotion.MC_AddAxisToGroup;
	{attribute 'hide'}
	fbRemoveAxisToGroup : Tc3_McCoordinatedMotion.MC_RemoveAxisFromGroup;
	{attribute 'hide'}
	fbGroupEnable 		: Tc3_McCoordinatedMotion.MC_GroupEnable;
	{attribute 'hide'}
	fbGroupDisable 		: Tc3_McCoordinatedMotion.MC_GroupDisable;
	{attribute 'hide'}
	fbGroupReadStatus 	: Tc3_McCoordinatedMotion.MC_GroupReadStatus;	
	{attribute 'hide'}
	fbUngroupAllAxes 	: Tc3_McCoordinatedMotion.MC_UngroupAllAxes;	
	{attribute 'hide'}
	fbGroupReset	 	: Tc3_McCoordinatedMotion.MC_GroupReset;
	{attribute 'hide'}
	nState_SEQ_Adding 	: UDINT;
	{attribute 'hide'}	
	fbMovers : CHALET_BaseComponents.FB_CH_List; // List of Axis to be added to the group
		
	//Link to CA Group
	GroupRef : AXES_GROUP_REF;
	
	{attribute 'hide'}	
	ipTempMover : I_XTS_Mover;

	{attribute 'hide'}
	dummyAxis : AXIS_REF;
	
	{attribute 'hide'}	
	fbFeedback : CHALET_BaseComponents.FB_CH_Feedback(ipSourceInfo := fbSourceInfo);
	
	{attribute 'hide'}
	eActiveCommand : E_NcGroupCommands := E_NcGroupCommands.None;

END_VAR

METHOD AddAxisListToGroup : HRESULT
VAR_INPUT
	ipMovers : CHALET_BaseComponents.I_CH_List;
END_VAR
IF NOT THIS^.fbFeedback.Done THEN
	//Errror active/not ready
	THIS^.fbFeedback.LastCommandAccepted := FALSE;
	
ELSIF nState_SEQ_Adding <> 0 AND nState_SEQ_Adding <> 999 THEN
	// Adding Sequence is not finished. Terminate first
	THIS^.fbFeedback.LastCommandAccepted := FALSE;

ELSIF ipMovers = 0 THEN
	// Invalide input
	THIS^.fbFeedback.LastCommandAccepted := FALSE;
		
ELSE
	// duplicate List
	THIS^.fbMovers.Duplicate(ipListCopyFrom := ipMovers);
	
	
	THIS^.nState_SEQ_Adding := 1;
	THIS^.fbFeedback.LastCommandAccepted := TRUE;
	THIS^.eActiveCommand := E_NcGroupCommands.AddAxisListToGroup;
	THIS^.fbFeedback.Busy := TRUE;	

END_IF

IF THIS^.fbFeedback.LastCommandAccepted THEN
	AddAxisListToGroup := S_OK;
ELSE
	AddAxisListToGroup := E_FAIL;
END_IF
END_METHOD

METHOD AddingAxisToGroup : HRESULT
VAR
	hr : HRESULT;
END_VAR
VAR_INST
	ipMover : CHALET_BaseComponents.I_CH_Object;
END_VAR
AddingAxisToGroup := S_PENDING;

CASE nState_SEQ_Adding OF
	0: // Idle
		AddingAxisToGroup := S_OK;
		
		
	1: // prepare List for iteratrion 
		THIS^.fbMovers.ResetIterator();
		nState_SEQ_Adding := 10;
		
		
	10: // has next Mover?
		IF THIS^.fbMovers.HasNextObject() THEN
			ipMover := THIS^.fbMovers.GetNextObject();
			IF ToMover(ipMover, ipTempMover) THEN
				nState_SEQ_Adding := 20;
			END_IF
		ELSE 
			nState_SEQ_Adding := 100;			
		END_IF
		
		
	20: // get Axis Reference
		IF ipTempMover <> 0 AND_THEN __ISVALIDREF(ipTempMover.getAxisRef) THEN
			nState_SEQ_Adding := 30;
		ELSE
			nState_SEQ_Adding := 1000 + nState_SEQ_Adding;	
		END_IF
		
		
	30: // add mover to group
		fbAddAxisToGroup.Execute := TRUE;
		IF fbAddAxisToGroup.Error THEN
			nState_SEQ_Adding := 1000 + nState_SEQ_Adding;
		ELSIF fbAddAxisToGroup.Done THEN
			nState_SEQ_Adding := 40;
			ipTempMover.MoverInGroup := TRUE;
		END_IF

	40: // Remove Object from List
		IF THIS^.fbMovers.RemoveObject(ipMover) THEN
			THIS^.fbMovers.ResetIterator();
			nState_SEQ_Adding := 10;
		ELSE
			nState_SEQ_Adding := 1000 + nState_SEQ_Adding;	
		END_IF
			
		
	100: // clear list
		// todo THIS^.iMovers.Clear();	
		nState_SEQ_Adding := 999;
		
		
	999: // Done
		AddingAxisToGroup := S_OK;

		
	1000..1999://Error
		hr := GetMostSignificant(hr, E_FAIL);	
			
END_CASE

// Propagate error
IF FAILED(hr) THEN
	AddingAxisToGroup := hr;
END_IF

// set feedback
THIS^.fbFeedback.HR := hr;
END_METHOD

PROPERTY AllAxesStanding : BOOL
GET
AllAxesStanding := fbGroupReadStatus.AllAxesStanding;
END_GET
END_PROPERTY

METHOD ChangeGapMode : HRESULT
VAR_INPUT
	bFast : BOOL;
END_VAR
ChangeGapMode := S_PENDING;

IF bFast THEN
	// Change fist to positive direction and then to Fast Mode	
	ipUtilityCAGroup.SetGapControlDirection(MC_GAP_CONTROL_DIRECTION.mcGapCtrlDirectionPositive);
	ipUtilityCAGroup.SetDefaultGapControlMode(MC_DEFAULT_GAP_CONTROL_MODE.mcGapCtrlModeFast);
ELSE
	// Change first to StandardMode and then to both direction
	ipUtilityCAGroup.SetDefaultGapControlMode(MC_DEFAULT_GAP_CONTROL_MODE.mcGapCtrlModeStandard);
	ipUtilityCAGroup.SetGapControlDirection(MC_GAP_CONTROL_DIRECTION.mcGapCtrlDirectionBoth);
END_IF

ChangeGapMode := S_OK;
END_METHOD

METHOD Disable : HRESULT
THIS^.fbFeedback.LastCommandAccepted := TRUE;
THIS^.fbFeedback.Busy := TRUE;	
THIS^.fbGroupDisable.Execute := TRUE;
THIS^.eActiveCommand := E_NcGroupCommands.GroupDisable;



IF THIS^.fbFeedback.LastCommandAccepted THEN
	Disable := S_OK;
ELSE
	Disable := E_FAIL;
END_IF
END_METHOD

METHOD Enable : HRESULT
IF NOT THIS^.fbFeedback.Done THEN
	THIS^.fbFeedback.LastCommandAccepted := FALSE;
	// Error active/not ready
	
ELSIF NOT(THIS^.fbGroupReadStatus.GroupDisabled) THEN
	THIS^.fbFeedback.LastCommandAccepted := FALSE;
	// Group in wrong State
	
ELSE
	THIS^.fbFeedback.LastCommandAccepted := TRUE;
	THIS^.fbFeedback.Busy := TRUE;
	THIS^.eActiveCommand := E_NcGroupCommands.GroupEnable;
	THIS^.fbGroupEnable.Execute := TRUE;
END_IF

IF THIS^.fbFeedback.LastCommandAccepted THEN
	Enable := S_OK;
ELSE
	Enable := E_FAIL;
END_IF
END_METHOD

METHOD FB_init : BOOL
VAR_INPUT
	bInitRetains : BOOL; // if TRUE, the retain variables are initialized (warm start / cold start)
	bInCopyCode : BOOL;  // if TRUE, the instance afterwards gets moved into the copy code (online change)
	
	ipXtsSystem : I_XTS_System_Registration; //Interface to XTS system object	
END_VAR
VAR_INST
	{attribute 'hide'}
	bFBInitCalledOnce : BOOL; //Do the following code once during start up and not during onlinechange
END_VAR
//Do the following code once during start up and not during onlinechange
IF NOT bFBInitCalledOnce THEN 
	
	//Regristrate object in System
	IF ipXtsSystem <> 0 THEN
		ipXtsSystem.LinkGroup(THIS^);
		THIS^.ipXtsSystem := ipXtsSystem;
	END_IF

END_IF

bFBInitCalledOnce := TRUE;
END_METHOD

{attribute 'monitoring':='call'}
PROPERTY GroupEnabled : BOOL
GET
GroupEnabled := fbGroupReadStatus.Valid AND NOT (fbGroupReadStatus.GroupDisabled OR fbGroupReadStatus.GroupErrorStop);
END_GET
END_PROPERTY

{attribute 'monitoring':='call'}
PROPERTY HR : HRESULT
GET
HR := fbFeedback.hr;
END_GET
END_PROPERTY

METHOD Initialize : HRESULT
VAR
	stVarInfo : __SYSTEM.VAR_INFO;
END_VAR
VAR_INST
	//This error cannot be reset. Requires a reset cold
	{attribute 'hide'}	
	fbInitError : FB_TcAlarm;
END_VAR
IF NOT THIS^.bInitDone THEN

	Initialize := S_PENDING;

	
	// Check if link to Group is mapped
	IF NcParameterlist.ERROR_IF_NC_AXIS_IS_NOT_MAPPED AND_THEN F_GetMappingStatus(ADR(THIS^.GroupRef.NcToPlc), SIZEOF(THIS^.GroupRef.NcToPlc)) <> EPlcMappingStatus.MS_Mapped THEN
		IF NOT fbInitError.bRaised THEN 
			//This error cannot be reset. Requires a reset cold
			fbInitError.CreateEx(stEventEntry := TC_EVENTS.CHALET_NC_Events.VariableLinkMissing, ipSourceInfo := THIS^.fbSourceInfo, bWithConfirmation := FALSE);
			stVarInfo := __VARINFO(GroupRef.NcToPlc);
			fbInitError.ipArguments.AddString(stVarInfo.Symbol);
			fbInitError.Raise(0);
		END_IF
		Initialize := E_FAIL;
		RETURN;
	END_IF
	
	
	// Check if link to Group is mapped
	IF NcParameterlist.ERROR_IF_NC_AXIS_IS_NOT_MAPPED AND_THEN F_GetMappingStatus(ADR(THIS^.GroupRef.PlcToNc), SIZEOF(THIS^.GroupRef.PlcToNc)) <> EPlcMappingStatus.MS_Mapped THEN
		IF NOT fbInitError.bRaised THEN 
			//This error cannot be reset. Requires a reset cold
			fbInitError.CreateEx(stEventEntry:= TC_EVENTS.CHALET_NC_Events.VariableLinkMissing, ipSourceInfo := THIS^.fbSourceInfo, bWithConfirmation := FALSE);
			stVarInfo := __VARINFO(GroupRef.PlcToNc);
			fbInitError.ipArguments.AddString(stVarInfo.Symbol);
			fbInitError.Raise(0);
		END_IF
		Initialize := E_FAIL;		
		RETURN;
	END_IF	


		
	IF THIS^.ipXtsSystem.Environment <> 0 THEN
		ipUtilityCAGroup := THIS^.ipXtsSystem.Environment.UtilityEnvirement.Mc2CaGroup(1);
	END_IF

	THIS^.bInitDone := TRUE;
ELSE
	
	Initialize := S_OK;

END_IF
END_METHOD

{attribute 'monitoring':='call'}
PROPERTY Mapped : BOOL //Project is mapped to NC (NcToPlc and PlcToNc)
GET
VAR
	bNcToPlcNotMapped 	: BOOL;
	bPlcToNcNotMapped 	: BOOL;
END_VAR
bNcToPlcNotMapped := F_GetMappingStatus(ADR(THIS^.GroupRef.NcToPlc), SIZEOF(THIS^.GroupRef.NcToPlc)) <> EPlcMappingStatus.MS_Mapped;
bPlcToNcNotMapped := F_GetMappingStatus(ADR(THIS^.GroupRef.PlcToNc), SIZEOF(THIS^.GroupRef.PlcToNc)) <> EPlcMappingStatus.MS_Mapped;

Mapped := NOT bNcToPlcNotMapped AND NOT bPlcToNcNotMapped;
END_GET
END_PROPERTY

{attribute 'monitoring':='call'}
PROPERTY OID : OTCID
GET
OID := GroupRef.NcToPlc.Common.GroupOID;
END_GET
END_PROPERTY

METHOD RemoveAxisFromGroup : HRESULT
VAR_INPUT
	ipMover	: I_XTS_Mover;
END_VAR
IF ipMover = 0 THEN
	THIS^.fbFeedback.LastCommandAccepted	:= FALSE;
	//Error no valid input
	
ELSE
	THIS^.eActiveCommand := E_NcGroupCommands.RemoveAxisFromGroup;
	THIS^.fbFeedback.LastCommandAccepted := TRUE;
	THIS^.fbFeedback.Busy := TRUE;

	fbRemoveAxisToGroup.IdentInGroup := ipMover.IdentInGroup;
	fbRemoveAxisToGroup.Execute := TRUE;
	ipMover.MoverInGroup := FALSE;
END_IF

IF THIS^.fbFeedback.LastCommandAccepted THEN
	RemoveAxisFromGroup := S_OK;
ELSE
	RemoveAxisFromGroup := E_FAIL;
END_IF
END_METHOD

METHOD Reset : HRESULT
THIS^.eActiveCommand := E_NcGroupCommands.GroupReset;
THIS^.fbFeedback.LastCommandAccepted := TRUE;
THIS^.fbFeedback.Busy := TRUE;	

THIS^.fbGroupReset.Execute := TRUE;

IF THIS^.fbFeedback.LastCommandAccepted THEN
	Reset := S_OK;
ELSE
	Reset := E_FAIL;
END_IF
END_METHOD

METHOD UngroupAllAxes : HRESULT
THIS^.eActiveCommand := E_NcGroupCommands.UngroupAllAxes;
THIS^.fbFeedback.LastCommandAccepted := TRUE;
THIS^.fbFeedback.Busy := TRUE;	

THIS^.nState_SEQ_Adding := 0;

THIS^.fbUngroupAllAxes.Execute := TRUE;


IF THIS^.fbFeedback.LastCommandAccepted THEN
	UngroupAllAxes := S_OK;
ELSE
	UngroupAllAxes := E_FAIL;
END_IF
END_METHOD

METHOD Update : HRESULT
// ********************** Refresh Group Information ***********************************************
fbGroupReadStatus(AxesGroup:=  THIS^.GroupRef, Enable:= TRUE);

// ********************** Set feedback depending on active command *******************************
IF THIS^.eActiveCommand <> E_NcGroupCommands.None THEN
	fbFeedback.ActiveCommand 	:= TO_STRING(THIS^.eActiveCommand);	
END_IF

CASE THIS^.eActiveCommand OF 
  E_NcGroupCommands.GroupDisable:
		fbFeedback.Busy 		:= fbGroupDisable.Busy;
		fbFeedback.Done 		:= fbGroupDisable.Done;
		fbFeedback.ErrorId 		:= fbGroupDisable.ErrorId;
  
  E_NcGroupCommands.GroupEnable:
		fbFeedback.Busy 		:= fbGroupEnable.Busy;
		fbFeedback.Done 		:= fbGroupEnable.Done;
		fbFeedback.ErrorId 		:= fbGroupEnable.ErrorId;
  
  E_NcGroupCommands.GroupReset:
		fbFeedback.Busy 		:= fbGroupReset.Busy;
		fbFeedback.Done 		:= fbGroupReset.Done;
		fbFeedback.ErrorId 		:= fbGroupReset.ErrorId;  
  
  E_NcGroupCommands.AddAxisListToGroup: 
		fbFeedback.Busy 		:= nState_SEQ_Adding > 0 AND nState_SEQ_Adding < 999;
		fbFeedback.Done 		:= nState_SEQ_Adding = 999; 
//		fbFeedback.ErrorId 		:= ;
  
  E_NcGroupCommands.RemoveAxisFromGroup:
		fbFeedback.Busy 		:= fbRemoveAxisToGroup.Busy;
		fbFeedback.Done 		:= fbRemoveAxisToGroup.Done;
		fbFeedback.ErrorId 		:= fbRemoveAxisToGroup.ErrorId;
  
  E_NcGroupCommands.UngroupAllAxes:
		fbFeedback.Busy 		:= fbUngroupAllAxes.Busy;
		fbFeedback.Done 		:= fbUngroupAllAxes.Done;
		fbFeedback.ErrorId 		:= fbUngroupAllAxes.ErrorId;
  
END_CASE

// **********************  Stop to execute commands on .done or .error ***************************
IF THIS^.fbFeedback.Done OR THIS^.fbFeedback.Error THEN
	THIS^.eActiveCommand 				:= E_NcGroupCommands.None;
END_IF


// **********************  Cyclic calls  *********************************************************
IF THIS^.ipTempMover <> 0 THEN
	fbAddAxisToGroup(AxesGroup := THIS^.GroupRef, Axis := THIS^.ipTempMover.getAxisRef, IdentInGroup := ipTempMover.IdentInGroup);
ELSE
	fbAddAxisToGroup(AxesGroup := THIS^.GroupRef, Axis := dummyAxis);
END_IF

fbRemoveAxisToGroup(AxesGroup := THIS^.GroupRef);
fbGroupEnable(AxesGroup := THIS^.GroupRef);
fbGroupDisable(AxesGroup := THIS^.GroupRef);
fbUngroupAllAxes(AxesGroup := THIS^.GroupRef);
fbGroupReset(AxesGroup := THIS^.GroupRef);

// ********************** Reset all Execution flags **********************************************
fbAddAxisToGroup.Execute := FALSE;
fbRemoveAxisToGroup.Execute := FALSE;
fbGroupEnable.Execute := FALSE;
fbGroupDisable.Execute := FALSE;
fbUngroupAllAxes.Execute := FALSE;
fbGroupReset.Execute := FALSE;


// todo hresult
END_METHOD

{attribute 'monitoring':='call'}
PROPERTY UtilityCAGroup : I_Mc2CaGroup
GET
UtilityCAGroup := THIS^.ipUtilityCAGroup;
END_GET
END_PROPERTY

END_FUNCTION_BLOCK

// COMPENENTs/Mover/ProductData/FB_XTS_ProductData
FUNCTION_BLOCK FB_XTS_ProductData EXTENDS FB_CH_Object IMPLEMENTS I_XTS_ProductData
VAR
	{attribute 'hide'}
	ipMover : I_XTS_Mover_PLC;
END_VAR

{attribute 'monitoring':='call'}
PROPERTY LinkedMover : I_XTS_Mover_PLC
GET
LinkedMover := ipMover;
END_GET
END_PROPERTY

METHOD LinkToMover : BOOL //it is not necessary to call this method. This is already done internally
VAR_INPUT
	ipMoverPlc : I_XTS_Mover_PLC;
END_VAR
THIS^.ipMover := ipMoverPlc;
END_METHOD

END_FUNCTION_BLOCK

// COMPENENTs/Mover/FB_XTS_Axis
{attribute 'no_explicit_call' := 'Do not call the body - Stick to OOP'}
FUNCTION_BLOCK FB_XTS_Axis EXTENDS CHALET_NC.FB_NcAxis
VAR
	{attribute 'hide'}
	fbMoveAbsoluteCA		: ARRAY [0..1] OF MC_MoveAbsoluteCA;//A second function block is always required to use the BufferMode. It is not possible to trigger a move function block with new parameters while it is active.
	{attribute 'hide'}
	fbHaltCA				: MC_HaltCA;
	{attribute 'hide'}
	nActiveMoveAbsCa 		: UINT;
END_VAR

METHOD HaltCA : I_CH_Feedback
VAR_INPUT
	fDeceleration          : LREAL;
    fJerk                  : LREAL;
    fGap                   : LREAL;
END_VAR
IF THIS^.Feedback.Error THEN
	THIS^.fbFeedback.LastCommandAccepted	:= FALSE;
	//Error active/not ready
		
ELSE
	THIS^.eActiveCommand 					:= CHALET_Nc.E_NcAxisCommands.HaltCA;
	THIS^.fbFeedback.LastCommandAccepted	:= TRUE;		
	THIS^.fbFeedback.Busy 					:= TRUE;
	                                    	
	THIS^.fbHaltCA.Execute					:= TRUE;
	THIS^.fbHaltCA.Gap						:= fGap;
	
	
	//Deceleration
	//If input = 0  then use default dynamics
	IF fDeceleration = 0.0 THEN
		THIS^.fbHaltCA.Deceleration := THIS^.fDefaultDeceleration;
	ELSE
		THIS^.fbHaltCA.Deceleration := fDeceleration;
	END_IF
	
	//Jerk
	//If input = 0  then use default dynamics
	IF fJerk = 0.0 THEN
		THIS^.fbHaltCA.Jerk := THIS^.fDefaultJerk;
	ELSE
		THIS^.fbHaltCA.Jerk := fJerk;
	END_IF

END_IF


HaltCA := THIS^.fbFeedback;
END_METHOD

{attribute 'TcRpcEnable':='1'} //call methode via OPC-UA conection
METHOD MoveAbsoluteCA  : I_CH_Feedback
VAR_INPUT
	fPosition		: LREAL;
	
	(* This value determines the minimum gap to the predecessor for Collision Avoidance. *)
	fGap			: LREAL;
	
	(* Use the default dynamics if input=0. 
	The default dynamics can be read and written via property and is initialized with the default values in the NC parameter list. *)
	fVelocity		: LREAL;
	
	(* Use the default dynamics if input=0. 
	The default dynamics can be read and written via property and is initialized with the default values in the NC parameter list. *)
	fAcceleration	: LREAL;
	
	(* Use the default dynamics if input=0. 
	The default dynamics can be read and written via property and is initialized with the default values in the NC parameter list. *)
	fDeceleration	: LREAL;
	
	(* Use the default dynamics if input=0. 
	The default dynamics can be read and written via property and is initialized with the default values in the NC parameter list. *)
	fJerk			: LREAL;
	
	(* Defines the direction of the movement (e.g. for a modulo axis). 
		input=0 = mcDirectionNonModulo*)
	eDirection	: Tc3_Mc3Definitions.MC_DIRECTION;
	
	(* Use the Aborting mode without buffering if input=0. 
	BufferModes:
		-MC_Aborting: Default mode without buffering. The command is executed immediately and interrupts any other command that may be running.
		-MC_Buffered: The command is executed once no other command is running on the axis. The previous movement continues until it has stopped. The following command is started from standstill. *)
	eBufferMode   : Tc3_Mc3Definitions.MC_BUFFER_MODE;
END_VAR
VAR
	nInactiveInstance : UINT;
END_VAR
IF THIS^.Feedback.Error THEN
	THIS^.fbFeedback.LastCommandAccepted	:= FALSE;
	//Error active/not ready

ELSIF NOT THIS^.BufferEmpty THEN		
	THIS^.fbFeedback.LastCommandAccepted	:= FALSE;
	//Buffer not ready to store next motion command	
	
ELSIF NOT((eBufferMode <> Tc3_Mc3Definitions.MC_BUFFER_MODE.mcAborting) OR (eBufferMode <> Tc3_Mc3Definitions.MC_BUFFER_MODE.mcBuffered)) THEN		
	THIS^.fbFeedback.LastCommandAccepted	:= FALSE;
	//only mcAborting and mcBuffered are available 	
	
ELSIF NOT(THIS^.Axis.Status.StandStill OR THIS^.Axis.Status.DiscreteMotion OR THIS^.Axis.Status.ContinuousMotion OR THIS^.Axis.Status.SynchronizedMotion) THEN		
	THIS^.fbFeedback.LastCommandAccepted	:= FALSE;
	//Axis in wrong State
	
ELSIF (eBufferMode <> Tc3_Mc3Definitions.MC_BUFFER_MODE.mcAborting) AND bNewBufferCommadThisCycle THEN		
	THIS^.fbFeedback.LastCommandAccepted	:= FALSE;
	//Buffer not ready to store next motion command		
	//Max send one buffered motion command each cycle	
	
ELSE
	//A second function block is always required to use the BufferMode. It is not possible to trigger a move function block with new parameters while it is active.
	IF THIS^.fbMoveAbsoluteCA[nActiveMoveAbsCA].Busy THEN
		nInactiveInstance := (THIS^.nActiveMoveAbsCa + 1)MOD 2;
	ELSE
		nInactiveInstance := THIS^.nActiveMoveAbsCa;
	END_IF
	
	THIS^.eActiveCommand 				:= E_NcAxisCommands.MoveAbsoluteCA;
	THIS^.fbFeedback.LastCommandAccepted:= TRUE;		
	THIS^.fbFeedback.Busy 				:= TRUE;
	
	THIS^.fbMoveAbsoluteCA[nInactiveInstance].ContinuousUpdate := TRUE;
	THIS^.fbMoveAbsoluteCA[nInactiveInstance].Execute		:= TRUE;
	THIS^.fbMoveAbsoluteCA[nInactiveInstance].Gap			:= fGap;
	THIS^.fbMoveAbsoluteCA[nInactiveInstance].Position		:= fPosition;
	THIS^.fbMoveAbsoluteCA[nInactiveInstance].Direction		:= eDirection;
	THIS^.fbMoveAbsoluteCA[nInactiveInstance].BufferMode 	:= eBufferMode;
	
	//If the currend command is a buffered movement, then set a flag.
	IF eBufferMode <> Tc3_Mc3Definitions.MC_BUFFER_MODE.mcAborting THEN
		THIS^.bNewBufferCommadThisCycle := TRUE;
	END_IF
	
	//Velocity
	//If input = 0  then use default dynamics
	IF fVelocity = 0.0 THEN
		THIS^.fbMoveAbsoluteCA[nInactiveInstance].Velocity := THIS^.fDefaultVelocity;
	ELSE
		THIS^.fbMoveAbsoluteCA[nInactiveInstance].Velocity := fVelocity;
	END_IF
	
	//Acceleration
	//If input = 0  then use default dynamics
	IF fAcceleration = 0.0 THEN
		THIS^.fbMoveAbsoluteCA[nInactiveInstance].Acceleration := THIS^.fDefaultAcceleration;
	ELSE
		THIS^.fbMoveAbsoluteCA[nInactiveInstance].Acceleration := fAcceleration;
	END_IF
	
	//Deceleration
	//If input = 0  then use default dynamics
	IF fDeceleration = 0.0 THEN
		THIS^.fbMoveAbsoluteCA[nInactiveInstance].Deceleration := THIS^.fDefaultDeceleration;
	ELSE
		THIS^.fbMoveAbsoluteCA[nInactiveInstance].Deceleration := fDeceleration;
	END_IF
	
	//Jerk
	//If input = 0  then use default dynamics
	IF fJerk = 0.0 THEN
		THIS^.fbMoveAbsoluteCA[nInactiveInstance].Jerk := THIS^.fDefaultJerk;
	ELSE
		THIS^.fbMoveAbsoluteCA[nInactiveInstance].Jerk := fJerk;
	END_IF

END_IF


MoveAbsoluteCA := THIS^.fbFeedback;
END_METHOD

METHOD Update  : HRESULT
// ********************** Do initialisation first ***********************************************
IF NOT bInitDone THEN
	Update := THIS^.Initialize();
	RETURN;
END_IF

// ********************** Set feedback depending on active command *******************************
CASE THIS^.eActiveCommand OF                                                                      
	E_NcAxisCommands.MoveAbsoluteCA:                                                              
		fbFeedback.Busy 		:= fbMoveAbsoluteCA[nActiveMoveAbsCa].Busy;                       
		fbFeedback.Done 		:= fbMoveAbsoluteCA[nActiveMoveAbsCa].Done;                       
		fbFeedback.ErrorId 		:= fbMoveAbsoluteCA[nActiveMoveAbsCa].ErrorID;  
       
	E_NcAxisCommands.HaltCA:                                                              
		fbFeedback.Busy 		:= fbHaltCA.Busy;                       
		fbFeedback.Done 		:= fbHaltCA.Done OR fbHaltCA.CommandAborted;                       
		fbFeedback.ErrorId 		:= fbHaltCA.ErrorID;            
END_CASE                                                                                          

// **********************  Cyclic call super Update  *********************************************
SUPER^.Update();
                                                                                                  
                                                                                                  
// **********************  Cyclic calls  *********************************************************
fbMoveAbsoluteCA[0](Axis := THIS^.Axis);                                                          
fbMoveAbsoluteCA[1](Axis := THIS^.Axis);                                                          
fbHaltCA(Axis := THIS^.Axis);
                                                                                                
                                                                                                  
// ********************** Reset all Execution flags **********************************************
fbMoveAbsoluteCA[0].Execute := FALSE;                                                             
fbMoveAbsoluteCA[1].Execute := FALSE;
fbHaltCA.Execute := FALSE;                                                                                                  

                                                                                                 
// ****************Get the acive instance. Stay at the last active.*******************************
IF fbMoveAbsoluteCA[0].Active THEN                                                                
	nActiveMoveAbsCa := 0;
ELSIF fbMoveAbsoluteCA[1].Active THEN
	nActiveMoveAbsCa := 1;
END_IF

//Return
Update := THIS^.fbFeedback.HR;
END_METHOD

END_FUNCTION_BLOCK

// COMPENENTs/Mover/FB_XTS_Mover
{attribute 'no_explicit_call' := 'Do not call the body - Stick to OOP'}
FUNCTION_BLOCK FB_XTS_Mover EXTENDS FB_CH_Object IMPLEMENTS I_XTS_Mover, I_XTS_Mover_PLC
VAR	
	//Link to NC
	Axis : FB_XTS_Axis;

	{attribute 'hide'}
	bInitDone : BOOL;
	{attribute 'hide'}
	ipXtsSystem : I_XTS_System_Registration;
	{attribute 'hide'}
	ipUtilityMover : I_TcIoXtsXpuMover;
	{attribute 'hide'}
	ipProductData : I_XTS_ProductData; //later the required interface of the tool or product can be queried via query interface
	{attribute 'hide'}
	ipParentStation : I_XTS_Station; //This is the station in which the Mover is currently standing or moving.	
	{attribute 'hide'}
	ipNextMover : I_XTS_Mover;
	{attribute 'hide'}
	sTargedStation : STRING;
	{attribute 'hide'}
	fLastCmdTargedPosition : LREAL; //the last commanded target position [mm]
	{attribute 'hide'}
	fLastCmdTargedVelocity : LREAL; //the last commanded target speed
	{attribute 'hide'}	
	fLastCmdTargedGap 	: LREAL; //the last commanded target gap
	{attribute 'hide'}
	bInGroup : BOOL;	
	{attribute 'hide'}	
	lrTrackLentgh 			: LREAL; //[mm]  Modulo
	{attribute 'hide'}
	fbFeedback 					: CHALET_BaseComponents.FB_CH_Feedback(ipSourceInfo := fbSourceInfo);;
	
END_VAR
VAR PERSISTENT
	fDrivenDistance : LREAL;
END_VAR

METHOD Disable : HRESULT
Axis.PowerOff();


//Show as feedback the state of the includet axis
fbFeedback.ActiveCommand := Axis.Feedback.ActiveCommand;
fbFeedback.LastCommandAccepted := Axis.Feedback.LastCommandAccepted;
fbFeedback.HR := Axis.Feedback.hr;


IF Axis.Feedback.LastCommandAccepted THEN
	Disable := S_OK;
ELSE  
	Disable := E_FAIL;;	
END_IF
END_METHOD

METHOD Enable : HRESULT
Axis.PowerOn();


//Show as feedback the state of the includet axis
fbFeedback.ActiveCommand := Axis.Feedback.ActiveCommand;
fbFeedback.LastCommandAccepted := Axis.Feedback.LastCommandAccepted;
fbFeedback.HR := Axis.Feedback.hr;


IF Axis.Feedback.LastCommandAccepted THEN
	Enable := S_OK;
ELSE  
	Enable := E_FAIL;;	
END_IF
END_METHOD

METHOD HaltCA : HRESULT
VAR_INPUT
END_VAR
Axis.HaltCA(
	fDeceleration:= 0, //use default
	fJerk:= 0, //use default
	fGap:= fLastCmdTargedGap);
	

//Show as feedback the state of the includet axis
fbFeedback.ActiveCommand := Axis.Feedback.ActiveCommand;
fbFeedback.LastCommandAccepted := Axis.Feedback.LastCommandAccepted;
fbFeedback.HR := Axis.Feedback.hr;


IF Axis.Feedback.LastCommandAccepted THEN
	HaltCA := S_OK;
ELSE  
	HaltCA := E_FAIL;;	
END_IF
END_METHOD

METHOD MoveAbsCA : HRESULT
VAR_INPUT
	fPosition	: LREAL := MC_INVALID;
	fVelocity	: LREAL := MC_INVALID;
	fGap		: LREAL := MC_DEFAULT;
	eDirection	: Tc3_Mc3Definitions.MC_DIRECTION;
END_VAR
Axis.MoveAbsoluteCA(
	fPosition:= fPosition, 
	fVelocity:= fVelocity, 
	fGap:= fGap, 
	fAcceleration:= 0, //Use Axis default
	fDeceleration:= 0, //Use Axis default
	fJerk:= 0, 			//Use Axis default
	eDirection := eDirection,
	eBufferMode:= Tc3_Mc3Definitions.MC_BUFFER_MODE.mcAborting);

THIS^.fLastCmdTargedVelocity := fVelocity;
THIS^.fLastCmdTargedPosition := fPosition;
THIS^.fLastCmdTargedGap := fGap;


//Show as feedback the state of the includet axis
fbFeedback.ActiveCommand := Axis.Feedback.ActiveCommand;
fbFeedback.LastCommandAccepted := Axis.Feedback.LastCommandAccepted;
fbFeedback.HR := Axis.Feedback.hr;


IF Axis.Feedback.LastCommandAccepted THEN
	MoveAbsCA := S_OK;
ELSE  
	MoveAbsCA := E_FAIL;;	
END_IF
END_METHOD

METHOD Reset : HRESULT
Axis.Reset();

//Show as feedback the state of the includet axis
fbFeedback.ActiveCommand := Axis.Feedback.ActiveCommand;
fbFeedback.LastCommandAccepted := Axis.Feedback.LastCommandAccepted;
fbFeedback.HR := Axis.Feedback.hr;


IF Axis.Feedback.LastCommandAccepted THEN
	Reset := S_OK;
ELSE  
	Reset := E_FAIL;;	
END_IF
END_METHOD

{attribute 'OPC.UA.DA.Property' := '1'}
{attribute 'monitoring':='call'}
PROPERTY DefaultAcceleration : LREAL
GET
DefaultAcceleration := THIS^.Axis.DefaultAcceleration;
END_GET
SET
THIS^.Axis.DefaultAcceleration := DefaultAcceleration;
END_SET
END_PROPERTY

{attribute 'OPC.UA.DA.Property' := '1'}
{attribute 'monitoring':='call'}
PROPERTY DefaultDeceleration : LREAL
GET
DefaultDeceleration := THIS^.Axis.DefaultDeceleration;
END_GET
SET
THIS^.Axis.DefaultDeceleration := DefaultDeceleration;
END_SET
END_PROPERTY

{attribute 'OPC.UA.DA.Property' := '1'}
{attribute 'monitoring':='call'}
PROPERTY DefaultJerk : LREAL
GET
DefaultJerk := THIS^.Axis.DefaultJerk;
END_GET
SET
THIS^.Axis.DefaultJerk := DefaultJerk;
END_SET
END_PROPERTY

{attribute 'monitoring':='call'}
PROPERTY SetAcceleration : LREAL
GET
SetAcceleration := THIS^.Axis.SetAcceleration;
END_GET
END_PROPERTY

{attribute 'monitoring':='call'}
PROPERTY SetVelocity : LREAL
GET
SetVelocity := THIS^.Axis.SetVelocity;
END_GET
END_PROPERTY

{attribute 'monitoring':='call'}
PROPERTY Coupled : BOOL
GET
Coupled := THIS^.Axis.Coupled;
END_GET
END_PROPERTY

{attribute 'monitoring':='call'}
PROPERTY DrivenDistance : LREAL
GET
DrivenDistance := fDrivenDistance;
END_GET
END_PROPERTY

{attribute 'monitoring':='call'}
PROPERTY Feedback : I_CH_Feedback
GET
Feedback := THIS^.fbFeedback;
END_GET
END_PROPERTY

PROPERTY getAxisRef : REFERENCE TO Tc2_MC2.AXIS_REF
GET
getAxisRef REF= THIS^.Axis.getAxisRef;
END_GET
END_PROPERTY

PROPERTY IdentInGroup : IDENT_IN_GROUP_REF
GET
IdentInGroup := UDINT_TO_IDENTINGROUP(THIS^.Axis.getAxisRef.NcToPlc.AxisId);
END_GET
END_PROPERTY

{attribute 'monitoring':='call'}
PROPERTY LagDistance : LREAL
GET
LagDistance := THIS^.Axis.LagDistance;
END_GET
END_PROPERTY

{attribute 'monitoring':='call'}
PROPERTY LastCmdTargedGap : LREAL
GET
LastCmdTargedGap := fLastCmdTargedGap;
END_GET
END_PROPERTY

{attribute 'monitoring':='call'}
PROPERTY LastCmdTargedPosition : LREAL
GET
LastCmdTargedPosition := fLastCmdTargedPosition;
END_GET
END_PROPERTY

{attribute 'monitoring':='call'}
PROPERTY LastCmdTargedVelocity : LREAL
GET
LastCmdTargedVelocity := fLastCmdTargedVelocity;
END_GET
END_PROPERTY

{attribute 'monitoring':='call'}
PROPERTY MoverInGroup : BOOL
GET
MoverInGroup := bInGroup;
END_GET
SET
bInGroup := MoverInGroup;
END_SET
END_PROPERTY

{attribute 'monitoring':='call'}
PROPERTY Moving : BOOL
GET
Moving := THIS^.Axis.Moving;
END_GET
END_PROPERTY

{attribute 'monitoring':='call'}
PROPERTY NextMover : I_XTS_Mover
GET
NextMover := ipNextMover;
END_GET
END_PROPERTY

{attribute 'monitoring':='call'}
PROPERTY OID : OTCID
GET
OID := THIS^.Axis.OID;
END_GET
END_PROPERTY

{attribute 'monitoring':='call'}
PROPERTY ParentStation : I_XTS_Station
GET
ParentStation := ipParentStation;
END_GET
SET
ipParentStation := ParentStation;
END_SET
END_PROPERTY

{attribute 'monitoring':='call'}
PROPERTY PositionOnTrack : LREAL
GET
//Round to 3 digits. If Axis is not enabled, use act position
IF THIS^.Axis.getAxisRef.Status.Disabled THEN
	PositionOnTrack := TO_LREAL(TRUNC(THIS^.Axis.ActPosModulo*1000))/1000;
ELSE
	PositionOnTrack := TO_LREAL(TRUNC(THIS^.Axis.SetPosModulo*1000))/1000;	
END_IF
END_GET
END_PROPERTY

{attribute 'monitoring':='call'}
PROPERTY TargedStation : STRING
GET
TargedStation := sTargedStation;
END_GET
SET
sTargedStation := TargedStation;
END_SET
END_PROPERTY

METHOD FB_init : BOOL
VAR_INPUT
	bInitRetains : BOOL; // if TRUE, the retain variables are initialized (warm start / cold start)
	bInCopyCode : BOOL;  // if TRUE, the instance afterwards gets moved into the copy code (online change)
	
	ipXtsSystem : I_XTS_System_Registration; //Interface to XTS system object
END_VAR
VAR_INST
	{attribute 'hide'}
	bFBInitCalledOnce : BOOL; //Do the following code once during start up and not during onlinechange
END_VAR
//Do the following code once during start up and not during onlinechange
IF NOT bFBInitCalledOnce THEN 
	

	//Regristrate object in System
	IF ipXtsSystem <> 0 THEN
		ipXtsSystem.RegisterMover(THIS^);
		THIS^.ipXtsSystem := ipXtsSystem;
	END_IF


	
END_IF

bFBInitCalledOnce := TRUE;
END_METHOD

(*The _ PLC interface provides the user with a simplified interface for commanding between the stations. Sometimes, however, this is not enough. 
Either you get the corresponding interface with the __Queryinterface or you can get full access with this property.*)
PROPERTY FullAccess : I_XTS_Mover
GET
FullAccess := (THIS^);
END_GET
END_PROPERTY

METHOD Initialize : HRESULT
VAR

END_VAR
fbFeedback.hr := S_OK;	

IF NOT THIS^.bInitDone THEN
	fbFeedback.ActiveCommand := 'Init';
	
	//Get Tracklength from system
	THIS^.lrTrackLentgh := THIS^.ipXtsSystem.TrackLength;
	
	
	//Validate Settings
	IF (lrTrackLentgh <= 0) THEN
		fbFeedback.hr := GetMostSignificant(fbFeedback.hr, E_FAIL);		
	END_IF
	

	//If only one mover is in project, then interface stays 0.
	IF THIS^.ipXtsSystem.Movers.Size > 1 THEN
		THIS^.ipNextMover := THIS^.ipXtsSystem.getMoverInFront(THIS^);
		//Validate Settings
		IF (ipNextMover = 0) THEN
			fbFeedback.hr := GetMostSignificant(fbFeedback.hr, E_FAIL);	
		END_IF
	ELSE
		THIS^.ipNextMover := 0;
	END_IF
	
	// Get XTS Utility mover object
	IF ipXtsSystem.Environment <> 0 THEN
		ipUtilityMover := ipXtsSystem.Environment.UtilityEnvirement.GetMoverInterfaceByAxisId(THIS^.getAxisRef.NcToPlc.AxisId);
		//Validate 
		IF (ipUtilityMover = 0) THEN
			fbFeedback.hr := GetMostSignificant(fbFeedback.hr, E_FAIL);	
		END_IF
	END_IF
	
	
	//InitAxis
	fbFeedback.hr := GetMostSignificant(fbFeedback.hr, Axis.Initialize());	

	bInitDone := CheckOk(fbFeedback.hr);
END_IF

Initialize := fbFeedback.hr;
END_METHOD

{attribute 'monitoring':='call'}
PROPERTY PUBLIC ProductData : I_XTS_ProductData
GET
ProductData := ipProductData;
END_GET
SET
// No change. Same interface is set again
IF ipProductData = ProductData THEN
	;//Noting
	
ELSE

	// If allready an interface is linked. Unlink
	IF ipProductData <> 0 THEN
		ipProductData.LinkToMover(0);
		ipProductData := 0;
	END_IF
	
	// Link and store new interface
	IF ProductData <> 0 THEN
		ProductData.LinkToMover(THIS^);
		ipProductData := ProductData;
	END_IF
END_IF
END_SET
END_PROPERTY

METHOD Update : HRESULT
VAR
	fDistanceThisCycle : LREAL;
END_VAR
VAR_INST
	fLastMoverPosition : LREAL;
END_VAR
// Total distance traveled by the mover
IF Axis.Moving THEN
	fDistanceThisCycle := ABS(Axis.SetPosModulo-fLastMoverPosition);
	IF fDistanceThisCycle > (THIS^.lrTrackLentgh*0.5) THEN
		fDistanceThisCycle := THIS^.lrTrackLentgh-fDistanceThisCycle;
	END_IF
	fDrivenDistance := fDrivenDistance + fDistanceThisCycle;
END_IF

fLastMoverPosition := Axis.SetPosModulo;

Axis.Update();

//Show as feedback the state of the includet axis
fbFeedback.ActiveCommand := Axis.Feedback.ActiveCommand;
fbFeedback.HR := Axis.Feedback.hr;
END_METHOD

{attribute 'monitoring':='call'}
PROPERTY UtilityMover : I_TcIoXtsXpuMover
GET
UtilityMover := ipUtilityMover;
END_GET
END_PROPERTY

END_FUNCTION_BLOCK

// COMPENENTs/Station/FB_XTS_Station
{attribute 'no_explicit_call' := 'Do not call the body - Stick to OOP'}
FUNCTION_BLOCK FB_XTS_Station EXTENDS FB_CH_Object IMPLEMENTS I_XTS_Station, I_XTS_Station_PLC
VAR
	{attribute 'hide'}
	bInitDone : BOOL;
	bErrorDuringFbInit : BOOL; // Not possible to reset
	{attribute 'hide'}
	ipXtsSystem 				: I_XTS_System_Registration;
	{attribute 'hide'}	
	ipStationInFront 			: I_XTS_Station;
	{attribute 'hide'}	
	ipStationBehinde 			: I_XTS_Station;
	{attribute 'hide'}
	bSuppressDynamicsChange		: BOOL; // Suppress to change the dynamic(Gap+velocity) of passing movers. This is usefull in startup
	{attribute 'hide'}
	fMoverGapAtExit 			: LREAL; // Every mover that leaves or passes the station gets this new gap as a target.
	{attribute 'hide'}
	fMoverVelocityAtExit		: LREAL; // Every mover that leaves or passes the station gets this new velo as a target.	 
	{attribute 'hide'}
	fPositionOnTrack 			: LREAL;
	{attribute 'hide'}
	nMoverQueueSize 			: UINT;
	{attribute 'hide'}
	bReadyToRecvMovers 			: BOOL := TRUE;;
	{attribute 'hide'}
	fTargetPosWindow			: LREAL := 0.05; //[mm]
	{attribute 'hide'}
	tTargetPosMonitoringTime	: TIME := T#0MS;
	{attribute 'hide'}	
	fTrackLentgh 				: LREAL; //[mm]  Modulo
	{attribute 'hide'}
	fbAssignedMovers 			: CHALET_BaseComponents.FB_CH_List;		// List of movers approaching the station
	{attribute 'hide'}
	fbFeedback 					: CHALET_BaseComponents.FB_CH_Feedback(ipSourceInfo := fbSourceInfo);
	{attribute 'hide'}	
	bMoversInPlace : BOOL;
	
	{attribute 'TcInitSymbol'}
	OIDStationInfo : OTCID; //OID of XtsStationInfo object to visualize in Viewer. 0 if not used.
	{attribute 'hide'}
	ipStationInfo : I_TcIoXtsInfoServerInfoStation;
	
	//Simulation
	{attribute 'hide'}
	fSimulationProcessDuration 	: LREAL; //[s]
	{attribute 'hide'}
	sSimulationTargedStation	: STRING; //LUID of the targed station to automatic send after the duration
	
	
	// ipXtsSystem Is Not Valid at this point, call the konstruktor again in the FB_Init
	{attribute 'hide'}
	fbTrigger 					: FB_XTS_Trigger(ipXtsSystem);
	{attribute 'hide'}
	fbSortedListMoversInQueue	: FB_XTS_Zone(ipXtsSystem);
	
	//Statistic
	{attribute 'hide'}
	fMoverPerMin				: LREAL;
	
END_VAR

METHOD ChangePos : HRESULT
VAR_INPUT
	fNewPosOnTrack : LREAL;
END_VAR
// new Position not allowed
IF fNewPosOnTrack <= THIS^.StationBehinde.PositionOnTrack OR 
   fNewPosOnTrack >= THIS^.StationsAhead.PositionOnTrack THEN
	// failed
	ChangePos := E_FAIL;
	RETURN;
END_IF

// change position when Station is empty
IF NOT THIS^.MoversInPlace THEN
	THIS^.fPositionOnTrack := fNewPosOnTrack;
	
	fbTrigger.PositionOnTrack := THIS^.fPositionOnTrack;
	
	// Move the zone 10mm forward to make sure, that an Mover who is enabled at x.01mm is still in range
	fbSortedListMoversInQueue.EndPositionOnTrack := LMOD(lr_Value:=(THIS^.PositionOnTrack + 10.0), lr_Arg:= THIS^.fTrackLentgh); 
	//The zone window is the full system, with one small exception, a window of 0.001mm after the end.  Start and end must not be identical
	fbSortedListMoversInQueue.StartPositionOnTrack := LMOD(lr_Value:=(fbSortedListMoversInQueue.EndPositionOnTrack  + 0.0001), lr_Arg:= THIS^.fTrackLentgh); 
	
	ChangePos := S_OK;
ELSE
	// wait untli station is empty
	ChangePos := S_FALSE;
END_IF
END_METHOD

{attribute 'monitoring':='call'}
PROPERTY CtsEmptySpaceInQueue : UDINT
GET
//Handle UINT Overflow
IF THIS^.fbAssignedMovers.Size >= THIS^.nMoverQueueSize THEN
	CtsEmptySpaceInQueue := 0;
ELSE 
	CtsEmptySpaceInQueue := THIS^.nMoverQueueSize - THIS^.fbAssignedMovers.Size;
END_IF
END_GET
END_PROPERTY

{attribute 'monitoring':='call'}
PROPERTY CtsMoversInQueue : UDINT
GET
CtsMoversInQueue := THIS^.fbAssignedMovers.Size;
END_GET
END_PROPERTY

(*The _ PLC interface provides the user with a simplified interface for commanding between the stations. Sometimes, however, this is not enough. 
Either you get the corresponding interface with the __Queryinterface or you can get full access with this property.*)
PROPERTY FullAccess : I_XTS_Station
GET
FullAccess := (THIS^);
END_GET
END_PROPERTY

{attribute 'monitoring':='call'}
//[mm] Every mover that leaves or passes the station gets this new gap as a target.
PROPERTY MoverGapAtExit : LREAL
GET
MoverGapAtExit := fMoverGapAtExit;
END_GET
SET
fMoverGapAtExit := MoverGapAtExit;
END_SET
END_PROPERTY

{attribute 'monitoring':='call'}
PROPERTY MoverQueueSize : UINT
GET
MoverQueueSize := THIS^.nMoverQueueSize;
END_GET
SET
THIS^.nMoverQueueSize := MoverQueueSize;
END_SET
END_PROPERTY

{attribute 'monitoring':='call'}
PROPERTY MoversInPlace : BOOL
GET
THIS^.Prepare();//Prepare time-critical information, if not already done


MoversInPlace := bMoversInPlace;
END_GET
END_PROPERTY

{attribute 'monitoring':='call'}
PROPERTY MoversInQueue : REFERENCE TO ARRAY [0..(XtsParameterlist.MAX_MOVER_PER_SYSTEM-1)] OF I_XTS_Mover_PLC // Return a sorted list of movers in this zone. Index 0 is the mover in Front.
GET
MoversInQueue REF= THIS^.fbSortedListMoversInQueue.MoversInZone;
END_GET
END_PROPERTY

{attribute 'monitoring':='call'}
PROPERTY MoverVelocityAtExit : LREAL //[mm/s] Every mover that leaves or passes the station gets this new velocity as a target.
GET
MoverVelocityAtExit := fMoverVelocityAtExit;
END_GET
SET
fMoverVelocityAtExit := MoverVelocityAtExit;
END_SET
END_PROPERTY

{attribute 'monitoring':='call'}
//[mm] from the beginning of the assigned track
PROPERTY PositionOnTrack : LREAL
GET
PositionOnTrack := fPositionOnTrack;
END_GET
END_PROPERTY

{attribute 'monitoring':='call'}
PROPERTY SuppressDynamicsChange : BOOL // Suppress to change the dynamic(Gap+velocity) of passing movers. This is usefull in startup
GET
SuppressDynamicsChange := bSuppressDynamicsChange;
END_GET
SET
bSuppressDynamicsChange := SuppressDynamicsChange;
END_SET
END_PROPERTY

{attribute 'monitoring':='call'}
//A time that is waited as soon as the mover is in the station (including the monitoring window) before “MoversInPlace” is set. e.g. used to stabilize the workpiece
PROPERTY TargetPosMonitoringTime : TIME
GET
TargetPosMonitoringTime := tTargetPosMonitoringTime;
END_GET
SET
tTargetPosMonitoringTime := TargetPosMonitoringTime;
END_SET
END_PROPERTY

{attribute 'monitoring':='call'}
//How many mm before the mover reaches the position is “MoversInPlace” set for the process. 
//This distance can also be set very large (e.g. 100mm) for moving past without stopping.
PROPERTY TargetPosWindow : LREAL
GET
TargetPosWindow := fTargetPosWindow;
END_GET
SET
fTargetPosWindow := TargetPosWindow;
END_SET
END_PROPERTY

{attribute 'monitoring':='call'}
PROPERTY ProcessSimulationActive : BOOL
GET
ProcessSimulationActive := THIS^.fSimulationProcessDuration > 0;
END_GET
END_PROPERTY

METHOD PROTECTED Simulation : HRESULT
VAR_INST
	tonSimulationDelay : TON;
END_VAR
//Automatic send mover to next station in Simulation
//If a valid time (>0seconds) is set and the configured destination station exists, then the movers will be sent away automatically after this time from now on.
tonSimulationDelay.IN 	:= THIS^.ipXtsSystem.Enabled AND THIS^.MoversInPlace AND THIS^.ProcessSimulationActive;
tonSimulationDelay.PT	:= LREAL_TO_TIME(THIS^.fSimulationProcessDuration*1000.0);
tonSimulationDelay();
IF tonSimulationDelay.Q THEN
	THIS^.SendMoversToStation(sTargedStation := THIS^.sSimulationTargedStation);
END_IF
END_METHOD

//If a valid time (>0seconds) is set and the configured destination station exists, then the movers will be sent away automatically after this time from now on.
METHOD SimulationMode : HRESULT
VAR_INPUT
	fProcessDuration 	: LREAL; //[s]
	sTargedStation		: STRING; //LUID of the targed station to automatic send after the duration
END_VAR
VAR
	ipStation	: I_CH_Object;
	bValideLUID : BOOL;
END_VAR
//Search LUID in Stationslist
ipStation := THIS^.ipXtsSystem.Stations.FindLUID(sTargedStation);
bValideLUID := (ipStation <> 0); 

IF (fProcessDuration > 0) AND bValideLUID THEN
	//Valide config
	THIS^.fSimulationProcessDuration 	:=	fProcessDuration;
	THIS^.sSimulationTargedStation 		:=	sTargedStation;
	SimulationMode := S_OK;
ELSE
	//Simulation disabled
	THIS^.fSimulationProcessDuration 	:=	0;
	THIS^.sSimulationTargedStation 		:=	'';
	SimulationMode := S_FALSE;
END_IF
END_METHOD

{attribute 'monitoring':='call'}
PROPERTY MoverPerMin : LREAL
GET
MoverPerMin := THIS^.fMoverPerMin;
END_GET
END_PROPERTY

METHOD PROTECTED UpdateStatistic : HRESULT
VAR
	nCycleTime_ns : UDINT;
END_VAR
VAR_INST
	tWaitForXTS, tWaitForProcess 	: LTIME;
	nMoverPassingStation			: UINT;
END_VAR
//Validate settings. STATISTIC_AVG_PERIOD must be >0
IF NOT TIME_TO_BOOL(XtsParameterlist.STATISTIC_AVG_PERIOD) THEN
	UpdateStatistic := E_FAIL;
	RETURN;
END_IF

//Get this task cycle time
nCycleTime_ns := TwinCAT_SystemInfoVarList._TaskInfo[THIS^.nTaskIndex].CycleTime(*100ns*) * 100;


//Depending on whether the station gives the start signal to the process or not, decide which of the two times should be incremented.
IF THIS^.MoversInPlace THEN
	tWaitForProcess := tWaitForProcess + UDINT_TO_LTIME(nCycleTime_ns);
ELSE
	tWaitForXTS 	:= tWaitForXTS + UDINT_TO_LTIME(nCycleTime_ns);
END_IF


//Check for mover who is passing the station
IF THIS^.fbTrigger.MoverDetected THEN
	nMoverPassingStation := nMoverPassingStation +1;
END_IF


//Once the period is reached. Evaluate and reset
IF (tWaitForProcess + tWaitForXTS) >= TIME_TO_LTIME(XtsParameterlist.STATISTIC_AVG_PERIOD) THEN
	
	//Calculate passing mover per minute
	THIS^.fMoverPerMin := TO_LREAL(nMoverPassingStation)*TIME_TO_LREAL(TIME#1M)/TIME_TO_LREAL(XtsParameterlist.STATISTIC_AVG_PERIOD);

	
	
	tWaitForProcess	:= LTIME#0NS;
	tWaitForXTS 	:= LTIME#0NS;
	nMoverPassingStation := 0;
END_IF
END_METHOD

METHOD PROTECTED UpdateUtilityStation : HRESULT //Utility InfoStation, used in XTS Viewer. All functionality packed into one method for easier overwriting
VAR
	aStopPositionsInfoStation : ARRAY[1..Tc3_XTS_Utility.TcIoXtsEnvironmentParameterList.MaxXtsStopPositionsPerStation] OF LREAL;
	//aPartIDs : ARRAY[1..Tc3_XTS_Utility.TcIoXtsEnvironmentParameterList.MaxXtsPartsPerXpu] OF OTCID;
	fLastStopPosition 		: LREAL;
	nLoopIndex 				: UINT;	
    ipMovers 				: CHALET_BaseComponents.I_CH_List;
	ipTempMover 			: I_XTS_Mover;
	nXpuNo 					: UINT;
	nMoverNo 				: UINT;
	pObject 				: ITComObject;
	sName 					: STRING;
END_VAR


VAR_INST
	bUtilityStationInitDone : BOOL;
	nOldMoverQueueSize 		: UINT := CHALET_BaseComponents.GVL_Datatypes.cMaxUint;
	fOldPositionOnTrack 	: LREAL;
	anBias 					: ARRAY[1..2] OF INT;
	bInverted 				: BOOL;
END_VAR
//Validate inputs
IF THIS^.OIDStationInfo = 0 OR ipXtsSystem.Environment = 0 THEN
	RETURN;
END_IF	


// Initalize
IF NOT bUtilityStationInitDone THEN
	//Get interface to utility station belongs to this station via OID
    FOR nLoopIndex := 1 TO ipXtsSystem.Environment.UtilityEnvirement.InfoServerTcIo(1).P_InfoStationCount DO
		IF 	ipXtsSystem.Environment.UtilityEnvirement.InfoServerTcIo(1).P_InfoStationOids[nLoopIndex] = THIS^.OIDStationInfo THEN
			THIS^.ipStationInfo := ipXtsSystem.Environment.UtilityEnvirement.InfoServerTcIo(1).InfoStationTcIo(nInfoStation:= nLoopIndex);
			EXIT;
		END_IF
	END_FOR	
	
	// calculate Position Offset
	IF THIS^.ipStationInfo <> 0 THEN			
		ipMovers := ipXtsSystem.Movers;
		ipMovers.ResetIterator();
		nLoopIndex := 0;	
		WHILE ipMovers.HasNextObject() DO
			nLoopIndex := nLoopIndex + 1;
			IF ToMover(ipMovers.GetNextObject(),ipTempMover) THEN
				//get Xpu Number by AxisId
				nXpuNo := ipXtsSystem.Environment.UtilityEnvirement.GetXpuNumberByAxisId(ipTempMover.getAxisRef.NcToPlc.AxisId);
				//get Mover Number by AxisId
				nMoverNo := ipXtsSystem.Environment.UtilityEnvirement.XpuTcIo(nXpuNo).GetMoverNumberByAxisId(ipTempMover.getAxisRef.NcToPlc.AxisId);
				//calculate Bias
				anBias[nLoopIndex] := LREAL_TO_INT(ipXtsSystem.Environment.UtilityEnvirement.XpuTcIo(nXpuNo).MoverTcIo(nMoverNo).GetPositionInfo().fPartPosition - ipTempMover.getAxisRef.NcToPlc.ModuloActPos);
				IF nLoopIndex = 2 THEN
					 EXIT;
				END_IF
			END_IF
		END_WHILE
		
		// Validate bias, check for inverted direction
		IF anBias[1] <> anBias[2] THEN
			bInverted := TRUE; 
			ipMovers.ResetIterator();
			nLoopIndex := 0;	
			WHILE ipMovers.HasNextObject() DO
				nLoopIndex := nLoopIndex + 1;
				IF ToMover(ipMovers.GetNextObject(),ipTempMover) THEN
					//get Xpu Number by AxisId
					nXpuNo := ipXtsSystem.Environment.UtilityEnvirement.GetXpuNumberByAxisId(ipTempMover.getAxisRef.NcToPlc.AxisId);
					//get Mover Number by AxisId
					nMoverNo := ipXtsSystem.Environment.UtilityEnvirement.XpuTcIo(nXpuNo).GetMoverNumberByAxisId(ipTempMover.getAxisRef.NcToPlc.AxisId);
					//calculate inverted Bias
					anBias[nLoopIndex] := LREAL_TO_INT(ipXtsSystem.TrackLength - ipXtsSystem.Environment.UtilityEnvirement.XpuTcIo(nXpuNo).MoverTcIo(nMoverNo).GetPositionInfo().fPartPosition - ipTempMover.getAxisRef.NcToPlc.ModuloActPos);
					IF nLoopIndex = 2 THEN
						 EXIT;
					END_IF
				END_IF	
			END_WHILE
		END_IF
		
		//Set unique station name
		FW_ObjMgr_GetObjectInstance(oid:= THIS^.OIDStationInfo , iid:= TC_GLOBAL_IID_LIST.IID_ITComObject, pipUnk:= ADR(pObject));
		IF pObject <> 0 THEN
			sName := THIS^.LUID;
			pObject.TcSetObjectName(ADR(sName));
			pObject.TcRelease();
		END_IF

	END_IF
	bUtilityStationInitDone := TRUE;
END_IF




// Update
// Configure/draw station in viewer on change
IF (THIS^.ipStationInfo <> 0) AND (THIS^.nMoverQueueSize <> nOldMoverQueueSize OR THIS^.fPositionOnTrack <> fOldPositionOnTrack) THEN	
	nOldMoverQueueSize := THIS^.nMoverQueueSize;
	fOldPositionOnTrack := THIS^.fPositionOnTrack;
	
	//aPartIDs :=  ipXtsSystem.Environment.UtilityEnvirement.XpuTcIo(1).P_PartOids ;
	THIS^.ipStationInfo.SetPartObjectIds(ipXtsSystem.Environment.UtilityEnvirement.XpuTcIo(1).P_PartOids);
	THIS^.ipStationInfo.SetIsEnabled(TRUE);

	
	// Draw stop position if gap between mover, given by station behind, is set
	IF (StationBehinde <> 0) AND (THIS^.nMoverQueueSize > 0) AND THIS^.nMoverQueueSize <= 25 THEN
		//Clear array
		MEMSET(ADR(aStopPositionsInfoStation), SIZEOF(aStopPositionsInfoStation), 0);
		//Fill array
		FOR nLoopIndex := 1 TO THIS^.nMoverQueueSize DO
			fLastStopPosition := (nLoopIndex-1)*StationBehinde.MoverGapAtExit;
			aStopPositionsInfoStation[(nLoopIndex)] := (fLastStopPosition);
		END_FOR
		IF NOT bInverted THEN
			//Start Position
			THIS^.ipStationInfo.SetStartPositionOnPart(MAX((fPositionOnTrack + anBias[1] - fLastStopPosition), 0)); ///zzz Todo. The InfoStation can not draw stations in the modulo area
			//End Pos
			THIS^.ipStationInfo.SetEndPositionOnPart(fPositionOnTrack + anBias[1]);
		ELSE
			//Start Position
			THIS^.ipStationInfo.SetStartPositionOnPart(ipXtsSystem.TrackLength - (fPositionOnTrack + anBias[1]));					
			//End Pos
			THIS^.ipStationInfo.SetEndPositionOnPart(MAX((ipXtsSystem.TrackLength - (fPositionOnTrack + anBias[1] - fLastStopPosition)), 0)); ///zzz Todo. The InfoStation can not draw stations in the modulo area
		END_IF
		//StopPositions
		THIS^.ipStationInfo.SetStopPositions(aStopPositionsInfoStation);

		//Override color if is set to transparent
		IF THIS^.ipStationInfo.GetStationColor() = 0 THEN
			THIS^.ipStationInfo.SetStationColor(nStationColor:= CHALET_BaseComponents.E_Colors_ARGB.Darkred);
		END_IF
	ELSE
		//Clear array
		MEMSET(ADR(aStopPositionsInfoStation), SIZEOF(aStopPositionsInfoStation), 0);	
		//StopPositions
		THIS^.ipStationInfo.SetStopPositions(aStopPositionsInfoStation);
		//Start Pos
		THIS^.ipStationInfo.SetStartPositionOnPart(nStartPositionOnPart := fPositionOnTrack + anBias[1]);
		//End Position
		THIS^.ipStationInfo.SetEndPositionOnPart(nEndPositionOnPart := fPositionOnTrack + anBias[1]);
	END_IF
	
	
	
	//Color Station depending on function:
	// Waitingstation green
	IF (FIND(THIS^.LUID,'wait')>0) OR (FIND(THIS^.LUID,'Wait')>0) OR (FIND(THIS^.LUID,'Warte')>0) OR (FIND(THIS^.LUID,'warte')>0) THEN
		THIS^.UtilityStationInfo.SetStationColor(nStationColor := CHALET_BaseComponents.E_Colors_ARGB.Green);
	
	// Dynamicstation blue
	ELSIF THIS^.MoverQueueSize = 0 THEN
		THIS^.UtilityStationInfo.SetStationColor(nStationColor := CHALET_BaseComponents.E_Colors_ARGB.Royalblue);	
    
	// Process station red
	ELSE
		THIS^.UtilityStationInfo.SetStationColor(nStationColor := CHALET_BaseComponents.E_Colors_ARGB.Red);			
	END_IF

END_IF
END_METHOD

{attribute 'monitoring':='call'}
PROPERTY UtilityStationInfo : I_TcIoXtsInfoServerInfoStation
GET
UtilityStationInfo := THIS^.ipStationInfo;
END_GET
END_PROPERTY

METHOD AddMoverToQueue : HRESULT
VAR_INPUT
	ipMover : I_XTS_Mover;
END_VAR
VAR
	ipObject : I_CH_Object;
END_VAR
//Get I_CH_Objekt of mover to put it in to a list.
IF ipMover <> 0 AND_THEN __QUERYINTERFACE(ipMover,ipObject) THEN
	//Add in List of Movers in this station
	THIS^.fbAssignedMovers.AddObject(ipObject);
	
	//Handover information in Mover
	ipMover.ParentStation := (THIS^);

	AddMoverToQueue := S_OK;
ELSE
	AddMoverToQueue := E_FAIL;;	
END_IF
END_METHOD

METHOD DeleteMoversQueue : HRESULT
VAR
	ipTempMover : I_XTS_Mover;
END_VAR
//Delete intormation in linked mover
fbAssignedMovers.ResetIterator();
WHILE fbAssignedMovers.HasNextObject() DO
	IF ToMover(fbAssignedMovers.GetNextObject(),ipTempMover) THEN
		ipTempMover.ParentStation := 0;
	END_IF	
END_WHILE

//Clear list
THIS^.fbAssignedMovers.Clear();
DeleteMoversQueue := S_OK;
END_METHOD

METHOD FB_init : BOOL
VAR_INPUT
	bInitRetains : BOOL; // if TRUE, the retain variables are initialized (warm start / cold start)
	bInCopyCode : BOOL;  // if TRUE, the instance afterwards gets moved into the copy code (online change)
	
	ipXtsSystem 			: I_XTS_System_Registration; //Interface to XTS system object
	fPositionOnTrack 		: LREAL;	//[mm]
	sUniqueName				: STRING;	//expl.:'Loading'
	nMoverQueueSize 		: UINT;		//[cts]
	
	//Dynamik at exit of station
	fMoverGapAtExit 		: LREAL;	//[mm]
	fMoverVelocityAtExit 	: LREAL;	//[mm/s]

END_VAR
VAR_INST
	{attribute 'hide'}
	bFBInitCalledOnce : BOOL; //Do the following code once during start up and not during onlinechange
END_VAR
//Do the following code once during start up and not during onlinechange
IF NOT bFBInitCalledOnce THEN 
	
	//Regristrate object in System
	IF ipXtsSystem <> 0 THEN
		ipXtsSystem.RegisterStation(THIS^);
		THIS^.ipXtsSystem := ipXtsSystem;
	END_IF

	//"" is maybe entered in an waiting or dynamic station and the name is not important
	IF sUniqueName <> '' THEN 
		THIS^.fbSourceInfo.sName := sUniqueName;
	ELSE
		sUniqueName := THIS^.fbSourceInfo.sName;
	END_IF
	
	THIS^.fMoverGapAtExit := fMoverGapAtExit;
	THIS^.fMoverVelocityAtExit := fMoverVelocityAtExit;
	THIS^.nMoverQueueSize := nMoverQueueSize;
	THIS^.fPositionOnTrack := fPositionOnTrack;
	
	THIS^.fbTrigger.FB_init(FALSE,FALSE, ipXtsSystem);
	THIS^.fbSortedListMoversInQueue.FB_init(FALSE,FALSE, ipXtsSystem);

END_IF

bFBInitCalledOnce := TRUE;
END_METHOD

{attribute 'monitoring':='call'}
PROPERTY HR : HRESULT
GET
HR := fbFeedback.hr;
END_GET
END_PROPERTY

METHOD Initialize : HRESULT
VAR
	nLoopIndex : UDINT;
	nNbOfStationsChecked : UDINT;
	ipThisStation, ipTempStation, ipStationInFrontTemp : I_XTS_Station;
	bErrorStationInFrontNotFound, bErrorStationBehindeNotFound : BOOL;
END_VAR
VAR_INST
	//This error cannot be reset. Requires a reset cold
	{attribute 'hide'}	
	fbInitError : FB_TcAlarm;
	{attribute 'hide'}	
	fbMissingInterfaceAlarm : FB_TcAlarm;
	{attribute 'hide'}	
	fbInvalideStationPositionAlarm : FB_TcAlarm;
END_VAR
ipThisStation := (THIS^);

//Check Error during FB_Init
IF THIS^.bErrorDuringFbInit THEN
	IF NOT fbInitError.bRaised THEN 
		//This error cannot be reset. Requires a reset cold
		fbInitError.CreateEx(stEventEntry:=TC_EVENTS.CHALET_Base_Events.ErrorFBinit, ipSourceInfo := THIS^.fbSourceInfo, bWithConfirmation := FALSE);
		fbInitError.Raise(0);
	END_IF
	Initialize:= E_FAIL;
	THIS^.fbFeedback.HR := Initialize;
	RETURN;
END_IF	

//Interface to System is missing
IF THIS^.ipXtsSystem = 0 THEN
	IF NOT fbMissingInterfaceAlarm.bRaised THEN 
		//This error cannot be reset. Requires a reset cold
		fbMissingInterfaceAlarm.CreateEx(stEventEntry:=TC_EVENTS.CHALET_XTS_Events.InitializationInvalideParameter, ipSourceInfo := THIS^.fbSourceInfo, bWithConfirmation := FALSE);
		fbMissingInterfaceAlarm.Raise(0);
	END_IF
	Initialize := E_FAIL;
	THIS^.fbFeedback.HR := Initialize;
	RETURN;
END_IF

//Station position on track is larger than CA-Group track length
IF THIS^.PositionOnTrack > THIS^.ipXtsSystem.TrackLength THEN
	IF NOT fbInvalideStationPositionAlarm.bRaised THEN 
		//This error cannot be reset. Requires a reset cold
		fbInvalideStationPositionAlarm.CreateEx(stEventEntry:=TC_EVENTS.CHALET_XTS_Events.StationPositionLargerAsTrack, ipSourceInfo := THIS^.fbSourceInfo, bWithConfirmation := FALSE);
		fbInvalideStationPositionAlarm.Raise(0);
	END_IF
	Initialize := E_FAIL;
	THIS^.fbFeedback.HR := Initialize;
	RETURN;
END_IF

//New Station in Front found. Befor continous do this for each station.
ipStationInFrontTemp := THIS^.ipXtsSystem.getStationInFront(THIS^);
IF ipStationInFrontTemp <> THIS^.ipStationInFront THEN
	THIS^.ipStationInFront := ipStationInFrontTemp;
	THIS^.bInitDone := FALSE;
	Initialize := S_PENDING;
	THIS^.fbFeedback.HR := Initialize;
	RETURN;
END_IF


fbFeedback.hr := S_OK;	

IF NOT THIS^.bInitDone THEN
	
	THIS^.DeleteMoversQueue();

	THIS^.fTrackLentgh := THIS^.ipXtsSystem.TrackLength;
	THIS^.ipStationInFront := THIS^.ipXtsSystem.getStationInFront(THIS^);
	
	
	fbTrigger.ListOfMoversToCheck := THIS^.ipXtsSystem.Movers;
	fbTrigger.PositionOnTrack := THIS^.PositionOnTrack;
	fbTrigger.TriggerDirection := MC_Positive_Direction;
	//Init Tigger
	fbFeedback.hr := GetMostSignificant(S_OK,fbTrigger.Initialize());	
	

	//Use the zone to sort all movers in this queue depending on the distance to targed in an output array.
	//The Zone is set to the length of the whole system, but only add the mover in the station queue.
	fbFeedback.hr := GetMostSignificant(fbFeedback.hr,fbSortedListMoversInQueue.Initialize());		
	// Move the zone 10mm forward to make sure, that an Mover who is enabled at x.01mm is still in range
	fbSortedListMoversInQueue.EndPositionOnTrack := LMOD(lr_Value:=(THIS^.PositionOnTrack + 10.0), lr_Arg:= THIS^.fTrackLentgh); 
	//The zone window is the full system, with one small exception, a window of 0.001mm after the end.  Start and end must not be identical
	fbSortedListMoversInQueue.StartPositionOnTrack := LMOD(lr_Value:=(fbSortedListMoversInQueue.EndPositionOnTrack  + 0.0001), lr_Arg:= THIS^.fTrackLentgh); 
	fbSortedListMoversInQueue.ListOfMoversToCheck := THIS^.fbAssignedMovers;
	fbFeedback.hr := GetMostSignificant(fbFeedback.hr,fbSortedListMoversInQueue.Initialize());		
	
	
	
	//Get Station behinde this one.
	ipTempStation := ipThisStation;
	nNbOfStationsChecked := 0;
	WHILE((ipTempStation <> 0) AND_THEN (ipTempStation.StationsAhead <> 0)) DO
		// test if this is the station behinde
		IF (ipTempStation.StationsAhead.LUID = THIS^.LUID) THEN
			THIS^.ipStationBehinde := ipTempStation;	
			EXIT;	
		END_IF
		// get Next Stations
		ipTempStation := ipTempStation.StationsAhead;
		nNbOfStationsChecked := nNbOfStationsChecked + 1;
		
		//Error, all station checked, not found.
		IF (ipTempStation = ipThisStation) OR (nNbOfStationsChecked > THIS^.ipXtsSystem.Stations.Size)THEN
			Initialize := E_FAIL;
			RETURN;
		END_IF
	END_WHILE

		
	//Validate Settings - Error
	bErrorStationInFrontNotFound := ((ipStationInFront = 0) AND THIS^.ipXtsSystem.Environment.TrackIsRing AND (THIS^.ipXtsSystem.Stations.Size > 1));
	bErrorStationBehindeNotFound := ((ipStationBehinde = 0) AND THIS^.ipXtsSystem.Environment.TrackIsRing AND (THIS^.ipXtsSystem.Stations.Size > 1));		
	IF (bErrorStationInFrontNotFound OR bErrorStationBehindeNotFound OR (THIS^.LUID = '') OR (fTrackLentgh <= 0) OR (fPositionOnTrack < 0.0) OR (fPositionOnTrack >= fTrackLentgh) OR (fMoverVelocityAtExit <= 0) OR (fMoverGapAtExit <= 0)) THEN
		fbFeedback.hr := GetMostSignificant(E_FAIL, fbFeedback.hr);	
		IF NOT fbInitError.bRaised THEN 
			//This error cannot be reset. Requires a reset cold
			fbInitError.CreateEx(stEventEntry:=TC_EVENTS.CHALET_XTS_Events.InitializationInvalideParameter, ipSourceInfo := THIS^.fbSourceInfo, bWithConfirmation := FALSE);
			fbInitError.Raise(0);
		END_IF
	END_IF

	
	bInitDone := CheckOk(fbFeedback.hr);
END_IF

				
								
Initialize := fbFeedback.hr;
END_METHOD

PROPERTY OID : OTCID
GET
OID := THIS^.OIDStationInfo;
END_GET
END_PROPERTY

(* 
	Use this Methode to calculate time sensitive date once each cycle. Example: read analog input and convert before do get Signal propertie
*)
METHOD PROTECTED Prepare : HRESULT
VAR_INST
	{attribute 'hide'}	
	nLastUpdatedCycleCount : UDINT;
END_VAR

VAR
	nLoopIndex : UINT;
	fExpectedDistanceToParent : LREAL;
	fPositionDifference : LREAL;
	nCycleTime_ms : UDINT;
	bMoverInQueue : BOOL;
	bTempMoverInPosition : BOOL;
	bTempMoverVeloZero : BOOL;
	bTempMoverInMonitoringTime : BOOL;
	bTempMoverThisStationAsTarged : BOOL;
END_VAR
VAR_INST
	{attribute 'hide'}
	nCycleCountInPos : UDINT;
END_VAR
//Check if this Cycle the dates are allready prepared. This is important for time sensitive informations.
IF nLastUpdatedCycleCount <> TwinCAT_SystemInfoVarList._TaskInfo[THIS^.TaskIndex].CycleCount THEN
	nLastUpdatedCycleCount := TwinCAT_SystemInfoVarList._TaskInfo[THIS^.TaskIndex].CycleCount ;


	(* Check if mover is in place. Time and Position window *)
	//If queuesize is zero, mover is never in place.
	IF nMoverQueueSize = 0 OR NOT ipXtsSystem.Enabled THEN
		THIS^.bMoversInPlace := FALSE;
		nCycleCountInPos := 0;
	ELSE
		//Get this task cycle Count and time 
		nCycleTime_ms := TwinCAT_SystemInfoVarList._TaskInfo[THIS^.nTaskIndex].CycleTime(*100ns*) / 10_000 ;
		
		bTempMoverInPosition := TRUE; bTempMoverVeloZero := TRUE; bTempMoverThisStationAsTarged := TRUE;
		fExpectedDistanceToParent := 0;
		FOR nLoopIndex := 0 TO (THIS^.nMoverQueueSize-1) DO
			IF THIS^.fbSortedListMoversInQueue.MoversInZone[nLoopIndex] <> 0 THEN
				//Check position and Gap - 1 mover do not have a gap
				IF nLoopIndex <> 0 THEN
					fExpectedDistanceToParent := fExpectedDistanceToParent + THIS^.fbSortedListMoversInQueue.MoversInZone[nLoopIndex].LastCmdTargedGap;
				END_IF
				bMoverInQueue		:= TRUE;
				
				fPositionDifference := F_GetDistToPosModulo(fTargedPosition := (THIS^.PositionOnTrack - fExpectedDistanceToParent),  fActualPosition :=  THIS^.fbSortedListMoversInQueue.MoversInZone[nLoopIndex].FullAccess.getAxisRef.NcToPlc.ModuloActPos, fModulo := THIS^.ipXtsSystem.TrackLength);
				IF fPositionDifference > (THIS^.ipXtsSystem.TrackLength/2) THEN
					fPositionDifference := (THIS^.ipXtsSystem.TrackLength - fPositionDifference);
				END_IF
				
				bTempMoverInPosition := bTempMoverInPosition AND (ABS(fPositionDifference) <= fTargetPosWindow );
				bTempMoverVeloZero := bTempMoverVeloZero AND (THIS^.fbSortedListMoversInQueue.MoversInZone[nLoopIndex].SetVelocity = 0);
				bTempMoverThisStationAsTarged := bTempMoverThisStationAsTarged AND ((THIS^.fbSortedListMoversInQueue.MoversInZone[nLoopIndex].TargedStation = THIS^.LUID));
			ELSE
				//Missing mover in queue
				bMoverInQueue := FALSE;
				EXIT;
			END_IF
		END_FOR
			
		//start time if mover position is ok
		IF bTempMoverInPosition  THEN
			nCycleCountInPos := nCycleCountInPos + 1;
		ELSE
			nCycleCountInPos := 0;
		END_IF
		
		bTempMoverInMonitoringTime := (UDINT_TO_TIME(nCycleCountInPos * nCycleTime_ms) >= tTargetPosMonitoringTime);
				
		THIS^.bMoversInPlace := bMoverInQueue AND bTempMoverInPosition AND bTempMoverInMonitoringTime AND bTempMoverThisStationAsTarged;// AND bTempMoverVeloZero;
	END_IF
	
	
END_IF
END_METHOD

{attribute 'monitoring':='call'}
//prevent further movers from entering the station, 
//e.g. to prevent a collision. All movers that are already moving to reach this station will be stopped with a stop 
//and restarted with Ready True.
PROPERTY ReadyToRecvMovers : BOOL
GET
ReadyToRecvMovers := bReadyToRecvMovers;
END_GET
SET
VAR
	ipTempMover : I_XTS_Mover;
END_VAR
//Change to Not Ready:
IF (ReadyToRecvMovers = FALSE) AND (bReadyToRecvMovers <> ReadyToRecvMovers) THEN
	//halt all movers on the way
	fbAssignedMovers.ResetIterator();
	WHILE fbAssignedMovers.HasNextObject() DO
		IF ToMover(fbAssignedMovers.GetNextObject(),ipTempMover) THEN
			ipTempMover.HaltCA();	
		END_IF	
	END_WHILE
END_IF

//Change to Ready:
IF (ReadyToRecvMovers = TRUE) AND (bReadyToRecvMovers <> ReadyToRecvMovers) THEN
	//all movers that are on the way have probably been stopped before. when reactivated, the last move command is sent again.
	fbAssignedMovers.ResetIterator();
	WHILE fbAssignedMovers.HasNextObject() DO
		IF ToMover(fbAssignedMovers.GetNextObject(),ipTempMover) THEN
			ipTempMover.MoveAbsCA(	fPosition	:= THIS^.PositionOnTrack, 
								fVelocity 	:= ipTempMover.LastCmdTargedVelocity,  
								fGap 		:= ipTempMover.LastCmdTargedGap,  
								eDirection 	:= Tc3_Mc3Definitions.MC_DIRECTION.mcDirectionPositive);	
		END_IF	
	END_WHILE
END_IF

//Store new status
bReadyToRecvMovers := ReadyToRecvMovers;
END_SET
END_PROPERTY

METHOD SendMoversToStation : HRESULT //Send all Queued movers away by changing the targed station destination
VAR_INPUT
	sTargedStation	: STRING;
END_VAR
VAR
	nLoopIndex 		: UINT;;
	ipMover	: I_XTS_Mover;
END_VAR
//Invalide targed
IF sTargedStation = '' THEN
	SendMoversToStation := E_FAIL;
	RETURN;
END_IF

//Movers have not reached station and can not send away until complet
IF NOT THIS^.MoversInPlace THEN
	SendMoversToStation := E_FAIL;
	RETURN;
END_IF

//Send all Queued movers away by changing the targed station destination
FOR nLoopIndex := 0 TO nMoverQueueSize-1 DO
	IF THIS^.MoversInQueue[nLoopIndex] <> 0 AND_THEN __QUERYINTERFACE(THIS^.MoversInQueue[nLoopIndex],ipMover) THEN
		ipMover.TargedStation := sTargedStation;		
	END_IF
END_FOR
END_METHOD

{attribute 'monitoring':='call'}
PROPERTY StationBehinde : I_XTS_Station
GET
StationBehinde := ipStationBehinde;
END_GET
END_PROPERTY

{attribute 'monitoring':='call'}
PROPERTY StationsAhead : I_XTS_Station
GET
StationsAhead := ipStationInFront;
END_GET
END_PROPERTY

//This sequence tries to transfer the mover to the next station in the direction of travel and checks whether the next station has space for it. 
//If the next station is a "dummy" that only changes the dynamics of the passing mover, this station is skipped and the next station is searched one ahead.
//If the station is fully occupied, no action is taken and a new search can be made in the next cycle.
METHOD PRIVATE TrySendMoverToNextStation : HRESULT
VAR_INPUT
	ipMover	: I_XTS_Mover;
	fVelocity : LREAL;
	fGap : LREAL;
END_VAR
VAR
	bStationIsOnlyForDynamicChanges : BOOL;
	bStationIsFull					: BOOL;
	bStationHanMoreMoverThanAllowed : BOOL;
	bStationHasAFreePlaceInQueue 	: BOOL;
	bStationIsTheTarged				: BOOL;
	bStationIsNotReadyToRecvMovers	: BOOL;
	
	ipMoverObject 		: I_CH_Object;
	ipTempStation 		: I_XTS_Station;	
	ipTargedStation 	: I_XTS_Station;

	nXpuNo 				: UINT;
	iMoverNo 			: UINT;
	stCommand 			: ST_TcIoXtsMoverCommand;	
END_VAR
//Invalide interface
IF ipMover = 0 THEN
	TrySendMoverToNextStation := E_FAIL;
	RETURN;
END_IF

//Mover is not in this Station.
IF __QUERYINTERFACE(ipMover,ipMoverObject) AND_THEN NOT THIS^.fbAssignedMovers.ObjectInList(ipMoverObject) THEN
	TrySendMoverToNextStation := E_FAIL;
	RETURN;
END_IF

//Send to actual Station is not supported
IF ipMover.TargedStation = THIS^.LUID THEN
	TrySendMoverToNextStation := E_FAIL;
	RETURN;
END_IF


ipTempStation := (THIS^);
//This sequence tries to transfer the mover to the next station in the direction of travel and checks whether the next station has space for it. 
//If the next station is a "dummy" that only changes the dynamics of the passing mover, this station is skipped and the next station is searched one ahead.
//If the station is fully occupied, no action is taken and a new search can be made in the next cycle.
WHILE (ipTargedStation=0) DO
	
	//get next station in flow direction
	ipTempStation := ipTempStation.StationsAhead;

	//All Stations around the XTS tested, Station not Found
	IF ipTempStation.LUID = THIS^.LUID THEN
		TrySendMoverToNextStation := E_FAIL;
		RETURN;
	END_IF

